(* CoDeSys 2.3 export: V4620699.EXP *)
(* Libraries: STANDARD.LIB 5.6.98 12:03:02, TcBase.lib 14.5.09 12:14:08, TcBaseMath.lib 27.7.04 12:07:56, TcCX1000System.lib 11.10.10 12:52:26, TcDrive.lib 25.1.17 09:42:28, TcEtherCAT.lib 30.11.16 19:52:18, TcIoFunctions.lib 27.1.17 17:22:22, TcMath.lib 23.9.04 15:15:30, TcMC.lib 27.7.15 08:51:38, TcNC.lib 10.10.08 17:55:34, TcNcDrive.lib 19.1.10 10:33:24, TcSystem.lib 7.6.16 11:01:22, TcTestAndSet.lib 23.2.09 12:50:08, TcUtilities.lib 3.2.16 16:08:58 *)

(* Task configuration *)
TASK Standard (PRIORITY := 0, INTERVAL := T#1ms);
PRG_STARTUP();
PRG_ERROR_WARNING_CTRLE();
PRG_VISU();
PRG_PROCESS();
PRG_STATION_WORK_ST1();
PRG_COLLISION_DETECTION();
PRG_VELOCITY_DETECTION();
PRG_HW_WORK_ST1();
PRG_HW_GENERAL();
END_TASK
TASK Ctrl_Panel (PRIORITY := 1, INTERVAL := T#100ms);
PRG_USB_IO_PANEL();
END_TASK

(* Global variable list: Constant_Variablen *)
VAR_GLOBAL CONSTANT
(*Constant variables Axis*)
	gciAxisZ_St1				:UINT:=1;
	gciAxisS_St1				:UINT:=2;
	gciAxisMax				:UINT:=2;

	gciStationSt1				:UINT:=1;

	(* developpement *)
	(*sRootPLC:STRING(255):='C:';*)
	(* machine *)
	cssRootPLC:STRING(255):='c:\';
	cssRootUSB:STRING(255):='d:\';
	(* HDD *)
	csiMaxFileLine:INT:=2230;
	csiMaxCharPerLine:INT:=135;
	(* Axis *)
	csiMaxAxisFileObj:INT:=50;
(* Visualisation number max page *)
	csiMaxPage:INT:=60;
	(* Profile *)
	csiMaxProfile:INT:=100;
	csiMaxProfileParameter:INT:=88;		(* BEF alt: 85 *) (* PUM alt: 78 *) (* PUM alt: 75 *) (* PUM alt: 61 *) (* PUM alt: 60 *) (* PUM alt: 53 *) (* IGS3 alt: 42 *)(* IGS2 alt: 38 *)(* IGS alt 36 *)
(* Page number definition *)
	gT_PageNumber:ST_VISUPAGENUMBER;
(* Anzahl maximal Wstk für Aufzeichnung *)
	ciMaxWP:INT:=100;
(* Max Anzahl Profilparameter *)
	ciMaxProfileParameter:INT:=1000;
(* Drehrichtung des Tellers *)
	gciModuloDirection:INT:=MC_Shortest_Way;

(* Skalierungswert für S Achse *)
	grScaleSAxis_Distance_SM:REAL:=966.0;
	grScaleSAxis_Speed_SM:REAL:=650;
	grMaxSAxis_Speed_SM:REAL:=8241.758;	(* Max Motor Drehzahl *)
	grScaleSAxis_Distance_L:REAL:=966.0;
	grScaleSAxis_Speed_L:REAL:=16;


	grMaxSAxis_Speed_L:REAL:=3000.0;		(* Max Motor Drehzahl *)	(* IGS angepasst *)
	grMaxSAxis_Speed_M:REAL:=6000.0;	(* Max Motor Drehzahl *)	(* IGS *)


(* ZUM LOESCHEN *)
	grScaleSAxis_Distance:REAL:=966.0;
	grScaleSAxis_Speed:REAL:=164;
	grMaxSAxis_Speed:REAL:=10000.0;			(* Max Motor Drehzahl *)
	grMaxSAxis_SpeedAllowed:REAL:=7000.0;	(* Max Motor Drehzal die für Maschine zugelassen ist *)
END_VAR

(* Global variable list: Globale_Variablen *)
VAR_GLOBAL
	QVisCtrl :ST_QVISCTRLE;(*~	(QVis) (InOut:2)	~*)
	T_ExchgParam :ST_QVIS_EXCHG_PARAM;(*~	(QVis) (InOut:2)	~*)
	T_VisuQVis:ST_QVIS;
	TProcess : ST_PROCESS;
	TStation_Work_St1 : ST_STATION;

(* Structure layer 2 *)
	T_CtrlePanel:ST_CTRLEPANEL;
	T_HDD:ST_HDD;
	T_NovRam : ST_NOVRAM;
(* StartUp *)
	T_StartUp:ST_STARTUP;
(* UPS *)
	T_CtrleUPS : ST_CTRLE_UPS;
	TStatusUPS:ST_UPSStatus;
(* Profile, 40 records ID for each Station *)
	T_Profile:ST_PROFILE;
(* TwinSAFE *)
	T_TwinSafeCtrleIN AT %I*:ST_TWINSAFE_CTRLE_IN;
	T_TwinSafeCtrleOUT AT %Q*:ST_TWINSAFE_CTRLE_OUT;
	T_TwinSafeIn AT %I*:ST_TWINSAFE_IN;
	T_TwinSafeOut AT %I*:ST_TWINSAFE_OUT;
	T_TwinSafeFBError AT %I*:ST_TWINSAFE_FB_ERROR;
	T_TwinSafe_Ctrle_Z_Axis_St1 AT %Q* : ST_TWINSAFE_DRIVE;
	T_TwinSafe_Status_Z_Axis_St1 AT %I* : ST_TWINSAFE_DRIVE;
	T_TwinSafe_Ctrle_S2_Axis_St1 AT %Q* : ST_TWINSAFE_DRIVE;		(* IGS *)
	T_TwinSafe_Status_S2_Axis_St1 AT %I* : ST_TWINSAFE_DRIVE;		(* IGS *)
	T_TwinSafe_Ctrle_S3_Axis_St1 AT %Q* : ST_TWINSAFE_DRIVE;		(* IGS *)
	T_TwinSafe_Status_S3_Axis_St1 AT %I* : ST_TWINSAFE_DRIVE;		(* IGS *)
	gT_SafetyStatus:ST_SAFETY_STATUS;

	T_Z_St1_Ctrle:ST_AXIS_CTRLE;
(* Static Error List *)
	T_ErrorList:ST_ERROR_LIST;	(* Static define Error List *)
(* Password *)
	T_Password:ST_PASSWORD;
(* Einrichtlampe *)
	TMachineLamp : ST_CYLINDER;
(* Control Button Start/Stop *)
	T_CtrleBtStartStop:ST_CTRLEBUTTON;
(* Kollisionsüberwachung *)
	TCollisionDetection:ST_COLLISION_DETECTION;
(* Status der Beckhoffklemmen und Kopplert *)
	T_TerminalState AT %I* :ST_TERMINAL_STATE;
(* Zähler für das Löschen der Vorwarnungen *)
	giDeleteMessageNumber: INT:=0;
	gcarAxisConfig		:ARRAY[1..gcIAxisMax] OF ST_EXCHG_PARAM_TEACHIN;
	gxHardwareOFF:BOOL;	(* Für Simulationszwecke ohne Hardware *)
	gxAxisOFF:BOOL;		(* Für Simulationszwecke wenn nur der Servocontroller der Z Achse fehlt und der Rest der Hardware vorhanden ist *)

(* Freigaben der Achsenbewegung mittels dem Joystick *)
	gxEnable_Joystick_Axis_Z:BOOL;
	gxReleaseEnableSwitch:BOOL;	(* Freigabe für Bewegung der Achsen mittels dem Zustimmschalter *)
	gxResetDataAnalysis_St1:BOOL;
	gxInitialStateActivated:BOOL;	(* Merker für Grundstellungsfahrt, ob dies ausgelöst wurde oder nicht *)
	gxAxisPositionSettled:BOOL;
	gxSetSpeedInMovement:BOOL;
	gxSetupFunctionActive:BOOL;
	gxAxisAbsolutMovementActive:BOOL;
	gxHandModeActive:BOOL;
	gxBlockSetQuality:BOOL;
	gxSpindelCalibrationONOFF_St1:BOOL;

	gT_PreWarning:ST_PREWARNING;

	gxAddInfeedZ:BOOL;
	gxSetPartQuality:BOOL;

	gxWP_Analyse_ActiveWork:BOOL;
	gxWP_Analyse_ActiveInfeed:BOOL;
	gxWP_Analyse_ActiveCentering:BOOL;
	gxWP_Analyse_ResetCentCountValue:BOOL;

	gdiSavePartQuality:DINT;

	gxMachineAutomodeActive_St1St2:BOOL;

(* Process Daten Aufzeichnung *)
	T_ProcessData_St1:ST_PROCESSDATA;

	gsDriveNameProcessData: STRING:='';

	gxBlockChangeMovementVisuActiveMessage:BOOL;

	gxSpindleOverloadError:BOOL;

	garRockerMeasureValue:ARRAY [1..200] OF REAL;
	grRockerMaxValue:REAL;
	grRockerMinValue:REAL;
	grRockerQuality:REAL;
	grRockerAmplitude:REAL;
	grRockerAmplitudeMin:REAL;
	grRockerAmplitudeMax:REAL;
	grRockerQualityMin:REAL;
	grRockerQualityMax:REAL;
	gdiRockerCountHC:DINT;
	gdiRockerCountHCTime:DINT;
	grRockerPosition:REAL;

	(* Globale Z Achsen Position *)
	grZ_LoadPos:REAL;
	grZ_WorkStartPos:REAL;
	grZ_WorkEndPos:REAL;

	gudiTorqueOverloadCounterValueSt1:UDINT;		(* IGS *)

	gxCentringActive:BOOL;						(* IGS3 *)
	gxOnlyCentringActive:BOOL;					(* IGS3 *)
	gxSuspensionONOFF:BOOL;					(* IGS3 *)

	garPositionEndProcCalc:ARRAY [1..1] OF REAL;
	garCentringEndProcCalc:ARRAY [1..1] OF REAL;
	gxZAxisVelocityCtrlActive:BOOL;
	gxZFollowDistanceError:BOOL;

	gxProcessCylindricalAreaActive:BOOL;
END_VAR

(* Global variable list: HW_IN_OUT *)
VAR_GLOBAL
(*++++++++++++++++++INPUT+++++++++++++++++++++++++++++*)
(*Local Inputs Schaltschrank*)
	IiAToolTorque_St1							AT%IB0		:INT;	(* Analoger Sensor für Drehmomentüberwachung für die Werkzeug Spindel *)
	IiASpeedServoDrive							AT%IB2		:INT;	(* Geschwindigkeitseinstellung der Achse Z1 *)
	IiAToolTorque2_St1							AT%IB4		:INT;	(* Analoger Sensor für Drehmomentüberwachung für die Werkzeug Spindel *)		(* IGS *)
	IiARes83										AT%IB6		:INT;	(* Reserve *)

	IxAirSupply									AT%IX8.0	:BOOL;	(* Ueberwacht den Mindestdruck des pneu.Netzes *)
	IxCabinDoorLocked							AT%IX8.1	:BOOL;	(* Kabinentüre (Sicherheitstüre) verriegelt *)
	IxStartButton									AT%IX8.2	:BOOL;	(* Externe Starttaste *)
	IxStopButton									AT%IX8.3	:BOOL;	(* Externe Stopptaste *)
	IxReleaseButton								AT%IX8.4	:BOOL;	(* Externe Freigabetaste für Energieversorgung *)
	IxRes105										AT%IX8.5	:BOOL;	(* Reserve *)
	IxJoystick_X_Plus								AT%IX8.6	:BOOL;	(* Joystick X Plus Jog Bewegung *)
	IxJoystick_X_Minus							AT%IX8.7	:BOOL;	(* Joystick X  negativ Ink Bewegung *)
	IxJoystick_Y_Plus								AT%IX9.0	:BOOL;	(* Joystick Z1 Achsenbewegung positiv *)
	IxJoystick_Y_Minus							AT%IX9.1	:BOOL;	(* Joystick Z1 Achsenbewegung negativ *)
	IxFuse24VDC_OK								AT%IX9.2	:BOOL;	(* Sicherungen 24VDC OK *)
	IxEnablingSwitchPlusButton						AT%IX9.3	:BOOL;	(* Zustimmschalter Plus Taste *)
	IxEnablingSwitchMinusButton					AT%IX9.4	:BOOL;	(* Zustimmschalter Minus Taste *)
	IxToolDeflection_St1							AT%IX9.5	:BOOL;	(* Überwachung der Werkzeug Auslenkung für die Werkzeug Spindel *)
	IxBrakeReleaseZ1Axis_St1						AT%IX9.6	:BOOL;	(* Sensor für Bremse gelöst bei der Z1 Achse (Hubachse) *)
	IxJoystick_WorkpieceClamp_ON_St1				AT%IX9.7	:BOOL;	(* Joystick für das einschalten der Werkstückfixierung *)
	IxJoystick_AirTable_ON						AT%IX10.0	:BOOL;	(* Joystick für das einschalten der Luft des Tisches	 *)
	IxJoystick_VaccumTable_ON					AT%IX10.1	:BOOL;	(* Joystick für das einschalten des Vakuums des Tisches *)
	IxUpperToolGuide_WorkpieceClamped_St1		AT%IX10.2	:BOOL;	(* Sensor für Überwachung der Werkstückfixierung *)
	IxToolSpindle_L_Connect_St1					AT%IX10.3	:BOOL;	(* Spindelkopf L angeschlossen-->Nur als Option vorgesehen: noch nichts unternehmen *)	(* INFO brauchts nicht, wird über Visu gemacht *)
	IxCylWPUnfixAtWorkPos_St1					AT%IX10.4	:BOOL;	(* Sensor für WstkEntspannen ist auf ArbeitsPosition *)							(* IGS3 *)
	IxToolDeflection2_St1							AT%IX10.5	:BOOL;	(* Überwachung der Werkzeug Auslenkung2 für die Werkzeug Spindel *)			(* IGS3 *)
	IxSuspenstionFilled							AT%IX10.6	:BOOL;	(* Sensor für Suspension ist gefüllt *)											(* IGS3 *)
	IxRes123										AT%IX10.7	:BOOL;	(* Reserve *)
	IxRes124										AT%IX11.0	:BOOL;	(* Reserve *)
	IxRes125										AT%IX11.1	:BOOL;	(* Reserve *)
	IxRes126										AT%IX11.2	:BOOL;	(* Reserve *)
	IxRes127										AT%IX11.3	:BOOL;	(* Reserve *)
	IxRes128										AT%IX11.4	:BOOL;	(* Reserve *)
	IxRes129										AT%IX11.5	:BOOL;	(* Reserve *)
	IxRes130										AT%IX11.6	:BOOL;	(* Reserve *)
	IxRes131										AT%IX11.7	:BOOL;	(* Reserve *)

	IxTorqueOverload_St1							AT%IX12.0	:BOOL;	(* Clock-->Signal induktiver Sensor für Drehmomentüberlast *)						(* IGS *)

(*++++++++++++++++++++++++++++
	Schnittstelle PLC to Safety Program:
++++++++++++++++++++++++++++*)
	IxTwinSafeQuickStopMaster1_1					AT%IX14.0	:BOOL;	(* QuickStop Achsen Mastermodul1_1 von TwinSAFE *)
	IxTwinSafeQuickStopMaster2_1					AT%IX14.1	:BOOL;	(* QuickStop Achsen Mastermodul2_1 von TwinSAFE *)							(* IGS *)
	IxTwinSafeQuickStopMaster2_2					AT%IX14.2	:BOOL;	(* QuickStop Achsen Mastermodul2_2 von TwinSAFE *)							(* IGS *)



(*++++++++++++++++++OUTPUT+++++++++++++++++++++++++++++*)
(*Local Outputs Schaltschrank*)
	QxCtrlLampStartButton							AT%QX0.0	:BOOL;	(* Kontroll LED externe Starttaste *)
	QxCtrlLampStopButton							AT%QX0.1	:BOOL;	(* Kontroll LED externe Stopptaste *)
	QxCtrlLampReleaseButton						AT%QX0.2	:BOOL;	(* Kotroll LED externe Freigabetaste für Energieversorgung *)
	QxCtrlLampAxesCurrentOff						AT%QX0.3	:BOOL;	(* Kontroll LED externe Ausschalttaste der Achsen Energieversorgung *)
	QxRes154									AT%QX0.4	:BOOL;	(* Reserve *)
	QxSignalLampGreen							AT%QX0.5	:BOOL;	(* Grüne Signallampe *)
	QxSignalLampRed							AT%QX0.6	:BOOL;	(* Rote Signallampe *)
	QxSignalLampYellow							AT%QX0.7	:BOOL;	(* Gelbe Signallampe *)
	QxCabinDoorLock								AT%QX1.0	:BOOL;	(* Verriegelungschalter der Kabinentüre, mit Magnetkraft *)
	QxSetupModeLamp							AT%QX1.1	:BOOL;	(* Gelbe Anzeige für den Einrichtbetrieb *)
	QxReadyToOperateMasterModul1				AT%QX1.2	:BOOL;	(* Betriebsbereitschaftsausgabe an Z1 *)
	QxEnablingSwitchVibration						AT%QX1.3	:BOOL;	(* Vibration des Zustimmschalter *)
	QxReadyToOperateMasterModul2				AT%QX1.4	:BOOL;	(* Betriebsbereitschaftsausgabe an S	ReadyToOperate to S *)					(* IGS *)
	QxMeasRangeTorqueSensor_St1				AT%QX1.5	:BOOL;	(* Drehmoment Sensor Bereichsumschaltung von 0-2Nm auf 0-0.5Nm Station 1 *)		(* IGS *)
	QxControlTorqueSensor_St1					AT%QX1.6	:BOOL;	(* Drehmoment Sensor Kontrollfunktion aktivieren Station 1 *)						(* IGS *)
	QxRes165									AT%QX1.7	:BOOL;	(* Reserve *)

	QxEnableQuickStopMasterModul1				AT%QX2.0	:BOOL;	(* Mastermodul für Z1 Achse aktivieren und einleiten des Schnellstop *)
	QxEnableQuickStopMasterModul2				AT%QX2.1	:BOOL;	(* Mastermodul für S Achse aktivieren und einleiten des Schnellstop *)				(* IGS *)
	QxCoolant_St1								AT%QX2.2	:BOOL;	(* Elektromagnetisches Ventil für Kühlmittel *)									(* IGS2 *)
	QxFastStrokeOn_St1							AT%QX2.3	:BOOL;	(* Schnellhub (Frequenzumformer) Ein *)										(* IGS2 *)
	QxRes214									AT%QX2.4	:BOOL;	(* Reserve *)
	QxRes215									AT%QX2.5	:BOOL;	(* Reserve *)
	QxRes216									AT%QX2.6	:BOOL;	(* Reserve *)
	QxRes217									AT%QX2.7	:BOOL;	(* Reserve *)
	QxRes218									AT%QX3.0	:BOOL;	(* Reserve *)
	QxRes219									AT%QX3.1	:BOOL;	(* Reserve *)
	QxRes220									AT%QX3.2	:BOOL;	(* Reserve *)
	QxRes221									AT%QX3.3	:BOOL;	(* Reserve *)
	QxRes222									AT%QX3.4	:BOOL;	(* Reserve *)
	QxRes223									AT%QX3.5	:BOOL;	(* Reserve *)
	QxRes224									AT%QX3.6	:BOOL;	(* Reserve *)
	QxRes225									AT%QX3.7	:BOOL;	(* Reserve *)

	QxMachineLamp								AT%QX4.0	:BOOL;	(* Maschinenleuchte *)
	QxRes201									AT%QX4.1	:BOOL;	(* Reserve *)
	QxRes202									AT%QX4.2	:BOOL;	(* Reserve *)
	QxRes203									AT%QX4.3	:BOOL;	(* Reserve *)

	QiAToolDeflection_SM_St1						AT%QB6	:INT;	(* Servoventil für Werkzeug Auslenkung der Werkzeug Spindel SM & M *)
	QiAToolTorqueHC_SM_St1						AT%QB8	:INT;	(* Servoventil für Drehmomentüberwachung HC des Spindelkopf SM *)		(* TODO löschen *)
	QiAToolTorqueOverload_SM_St1				AT%QB10	:INT;	(* Servoventil für Werkzeug Auslenkung der Werkzeug Spindel L *)		(* ALT: Servoventil für Drehmomentüberwachung Überlast des Spindelkopf SM *)
	QiAFastStroke								AT%QB12	:INT;	(* Analog Ausgang für FU (Schnellhub) *)										(* IGS2 *)
	QiARes254									AT%QB14	:INT;	(* Reserve *)
	QiARes255									AT%QB16	:INT;	(* Reserve *)
	QiARes256									AT%QB18	:INT;	(* Reserve *)
	QiARes257									AT%QB20	:INT;	(* Reserve *)

(* External Outputs at SMC Valve Block  *)
	Qby0ValveBlock								AT%QB30	:BYTE;	(* Byte 0 for Ethercat ValveBlock, Contains all following BOOL-Vars *)
	QxCylBrakeReleaseZAxis_Open_St1				AT%QX30.0	:BOOL;	(* Ventil für Bremszylinder der Z1 Achse für Bremse lösen *)
	QxCylBrakeReleaseZAxis_Close_St1			AT%QX30.1	:BOOL;	(* Ventil für Bremszylinder der Z1 Achse für Bremse aktivieren *)
	QxCylWorkpieceClamp_St1						AT%QX30.2	:BOOL;	(* Ventil für Werkstückfixierzylinder *)
	QxRes303									AT%QX30.3	:BOOL;	(* Reserve *)
	QxAirTable									AT%QX30.4	:BOOL;	(* Ventil für die Luft des Tisches *)
	QxRes305									AT%QX30.5	:BOOL;	(* Reserve *)
	QxVacuumTable								AT%QX30.6	:BOOL;	(* Ventil für das Vakuum des Tisches *)
	QxRes307									AT%QX30.7	:BOOL;	(* Reserve *)

	Qby1ValveBlock								AT%QB31	:BYTE;	(* Byte 1 for Ethercat ValveBlock, Contains all following BOOL-Vars *)
	QxCylWPUnfix_St1							AT%QX31.0	:BOOL;	(* Ventil für ZylWstkEntspannen *)											(* IGS3 *)
	QxRes309									AT%QX31.1	:BOOL;	(* Reserve *)
	QxCylStripperClose_St1						AT%QX31.2	:BOOL;	(* Ventil für ZylAbstreiferGeschlossen *)										(* IGS3 *)
	QxCylStripperOpen_St1						AT%QX31.3	:BOOL;	(* Ventil für ZylAbstreiferOffen *)												(* IGS3 *)
	QxRes312									AT%QX31.4	:BOOL;	(* Reserve *)
	QxRes313									AT%QX31.5	:BOOL;	(* Reserve *)
	QxRes314									AT%QX31.6	:BOOL;	(* Reserve *)
	QxRes315									AT%QX31.7	:BOOL;	(* Reserve *)

	Qby2ValveBlock								AT%QB32	:BYTE;	(* Byte 2 for Ethercat ValveBlock, Contains all following BOOL-Vars *)
	QxRes316									AT%QX32.0	:BOOL;	(* Reserve *)
	QxRes317									AT%QX32.1	:BOOL;	(* Reserve *)
	QxRes318									AT%QX32.2	:BOOL;	(* Reserve *)
	QxRes319									AT%QX32.3	:BOOL;	(* Reserve *)
	QxRes320									AT%QX32.4	:BOOL;	(* Reserve *)
	QxRes321									AT%QX32.5	:BOOL;	(* Reserve *)
	QxRes322									AT%QX32.6	:BOOL;	(* Reserve *)
	QxRes323									AT%QX32.7	:BOOL;	(* Reserve *)

(*++++++++++++++++++++++++++++
	Schnittstelle PLC to Safety Program:
++++++++++++++++++++++++++++*)
	QxTwinSafeReleaseButton						AT%QX35.0	:BOOL;	(* Output to safety prog *)
	QxTwinSafeServoDrivesRdy					AT%QX35.1	:BOOL;	(* Output to safety prog,ALL Servo-Controler: No Error *)

END_VAR

(* Global variable list: TwinCAT_Configuration *)
(* Generated automatically by TwinCAT - (read only) *)
VAR_CONFIG
	PRG_HW_WORK_ST1.IuiActualTorqueAxisZ_St1 AT %IB1656 : UINT;
	PRG_HW_WORK_ST1.IwInputState_Z_Axis_St1 AT %IB1658 : WORD;	(*  ~ {LinkedWith:TIID^Gerät 4 (EtherCAT)^Achse Z St1 (AX5106-0000-0210)^AT^Digital inputs, state} *)
	PRG_HW_WORK_ST1.IuiActualTorqueAxisS_St1 AT %IB1660 : UINT;
	PRG_HW_WORK_ST1.IwInputState_S1_Axis_St1 AT %IB1662 : WORD;
	PRG_HW_WORK_ST1.IwInputState_S2_Axis_St1 AT %IB1012 : WORD;	(*  ~ {LinkedWith:TIID^Gerät 4 (EtherCAT)^Antrieb S2 S3 St1 (AX5206-0000-0203)^AT 1^Digital inputs, state} *)
	PRG_HW_WORK_ST1.IwInputState_S3_Axis_St1 AT %IB1014 : WORD;	(*  ~ {LinkedWith:TIID^Gerät 4 (EtherCAT)^Antrieb S2 S3 St1 (AX5206-0000-0203)^AT 2^Digital inputs, state} *)
	PRG_HW_WORK_ST1.stZRefIn_St1 AT %IB1016 : NCTOPLC_AXLESTRUCT;	(*  ~ {LinkedWith:TINC^NC-Task 1 SAF^Achsen^Achse Z^Ausgänge^Achse Z_ToPlc} *)
	PRG_HW_WORK_ST1.stZRefOut_St1 AT %QB10012 : PLCTONC_AXLESTRUCT;	(*  ~ {LinkedWith:TINC^NC-Task 1 SAF^Achsen^Achse Z^Eingänge^Achse Z_FromPlc} *)
	PRG_HW_WORK_ST1.stZDriveState_St1 AT %IB1144 : ST_AXIS_DRIVESTATE;
	PRG_HW_WORK_ST1.stSRefIn_St1 AT %IB1148 : NCTOPLC_AXLESTRUCT;	(*  ~ {LinkedWith:TINC^NC-Task 1 SAF^Achsen^Achse S1^Ausgänge^Achse S1_ToPlc} *)
	PRG_HW_WORK_ST1.stSRefOut_St1 AT %QB10140 : PLCTONC_AXLESTRUCT;	(*  ~ {LinkedWith:TINC^NC-Task 1 SAF^Achsen^Achse S1^Eingänge^Achse S1_FromPlc} *)
	PRG_HW_WORK_ST1.stS2RefIn_St1 AT %IB1276 : NCTOPLC_AXLESTRUCT;	(*  ~ {LinkedWith:TINC^NC-Task 1 SAF^Achsen^Achse S2^Ausgänge^Achse 2_ToPlc} *)
	PRG_HW_WORK_ST1.stS2RefOut_St1 AT %QB10268 : PLCTONC_AXLESTRUCT;	(*  ~ {LinkedWith:TINC^NC-Task 1 SAF^Achsen^Achse S2^Eingänge^Achse 2_FromPlc} *)
	PRG_HW_WORK_ST1.stS3RefIn_St1 AT %IB1404 : NCTOPLC_AXLESTRUCT;	(*  ~ {LinkedWith:TINC^NC-Task 1 SAF^Achsen^Achse S3^Ausgänge^Achse 3_ToPlc} *)
	PRG_HW_WORK_ST1.stS3RefOut_St1 AT %QB10396 : PLCTONC_AXLESTRUCT;	(*  ~ {LinkedWith:TINC^NC-Task 1 SAF^Achsen^Achse S3^Eingänge^Achse 3_FromPlc} *)
	PRG_HW_WORK_ST1.stBubblerDataINSt1 AT %IB1648 : ST_COMM_IN_DCAXIS;
	PRG_HW_WORK_ST1.stBubblerDataOUTSt1 AT %QB10587 : ST_COMM_OUT_DCAXIS;
	PRG_HW_WORK_ST1.stFeedpumpINDataSt1 AT %IB1651 : ST_COMM_IN_DCAXIS;
	PRG_HW_WORK_ST1.stFeedpumpOUTDataSt1 AT %QB10590 : ST_COMM_OUT_DCAXIS;
	PRG_HW_WORK_ST1.IudiTorqueOverloadCounterValue_St1 AT %IB1532 : UDINT;	(*  ~ {LinkedWith:TIID^Gerät 1 (EtherCAT)^E-CAT Netzteil  (EK1200)^Zaehlerklemme 15 (EL1502)^CNT Inputs^Counter value} *)
	PRG_USB_IO_PANEL.IarxCtrlePanelButton AT %IB1536 : ARRAY [1..10] OF BOOL;
	PRG_USB_IO_PANEL.QarxCtrlePanelLed AT %QB10524 : ARRAY [1..10] OF BOOL;
	.T_TwinSafeCtrleIN AT %IB1546 : ST_TWINSAFE_CTRLE_IN;
	.T_TwinSafeCtrleOUT AT %QB10534 : ST_TWINSAFE_CTRLE_OUT;
	.T_TwinSafeIn AT %IB1549 : ST_TWINSAFE_IN;
	.T_TwinSafeOut AT %IB1569 : ST_TWINSAFE_OUT;
	.T_TwinSafeFBError AT %IB1577 : ST_TWINSAFE_FB_ERROR;
	.T_TwinSafe_Ctrle_Z_Axis_St1 AT %QB10536 : ST_TWINSAFE_DRIVE;
	.T_TwinSafe_Status_Z_Axis_St1 AT %IB1585 : ST_TWINSAFE_DRIVE;
	.T_TwinSafe_Ctrle_S2_Axis_St1 AT %QB10553 : ST_TWINSAFE_DRIVE;
	.T_TwinSafe_Status_S2_Axis_St1 AT %IB1602 : ST_TWINSAFE_DRIVE;
	.T_TwinSafe_Ctrle_S3_Axis_St1 AT %QB10570 : ST_TWINSAFE_DRIVE;
	.T_TwinSafe_Status_S3_Axis_St1 AT %IB1619 : ST_TWINSAFE_DRIVE;
	.T_TerminalState AT %IB1636 : ST_TERMINAL_STATE;
END_VAR

(* Data type in Axis/Axis_DC_KL2552 *)
TYPE ST_AXIS_FILE_OBJ_DCAXIS :
STRUCT
	sData: ARRAY[1..csiMaxAxisFileObj] OF STRING(80);
END_STRUCT
END_TYPE

(* Data type in Axis/Axis_DC_KL2552 *)
TYPE ST_COMM_IN_DCAXIS :
STRUCT
	usiStatusWord :USINT;
	iDataIn :INT;
END_STRUCT
END_TYPE

(* Data type in Axis/Axis_DC_KL2552 *)
TYPE ST_COMM_OUT_DCAXIS :
STRUCT
	usiControlWord :USINT;
	iDataOut :INT;
END_STRUCT
END_TYPE

(* Data type in Axis/Axis_DC_KL2552 *)
TYPE ST_CONFIG_GENERAL_DCAXIS :
STRUCT
	sDeviceName:STRING(32);
	sDeviceFileName:STRING(32);
	sServoNetId:STRING(23);		(* Beckhoff *)
	udiNodeId:UDINT;				(* Maxon *)
	iTyp:INT;
	lrScaleFactor:LREAL:=0.0;
	lrInitFactor:LREAL:=0.0;
END_STRUCT
END_TYPE

(* Data type in Axis/Axis_DC_KL2552 *)
TYPE ST_CONFIG_OBJECT_DCAXIS :
STRUCT
	diMaxMotorCurrent:DINT:=0;
	diNominalMotorCurrent:DINT:=0;
	diMotorResistor:DINT:=0;
	diKpSpeedControl:DINT:=0;
	diTnCurrentControl:DINT:=0;
	diMaxTorqueMotor:DINT:=0;
	xSpeedControlAcitv:BOOL:=FALSE;
	xCurrentControlAcitv:BOOL:=FALSE;
	xWinCurrentControlActiv:BOOL:=FALSE;
	xTorqueControlAcitv:BOOL:=FALSE;
	xOverVoltageActiv:BOOL:=FALSE;
END_STRUCT
END_TYPE

(* Data type in Axis/Axis_DC_KL2552 *)
TYPE ST_CTRLE_DCAXIS :
STRUCT
(* Input *)
	xExecute:BOOL:=FALSE;
	iFunction:INT:=0;
	xReset:BOOL:=FALSE;
	lrVelocity:LREAL:=0;
	tAcceleration:TIME:=T#0s;
	tDecceleration:TIME:=T#0s;
	iRegisterNr:INT:=0;
	iValueRegister:INT:=0;

(* Output *)
	xDone:BOOL:=FALSE;
	xErr:BOOL:=FALSE;
	udiErrorID:UDINT:=0;
	xPower:BOOL:=FALSE;
	xReady:BOOL:=FALSE;
	xNotMoving:BOOL:=FALSE;
END_STRUCT
END_TYPE

(* Data type in Axis/Axis_DC_KL2552 *)
TYPE ST_DC_AXIS :
STRUCT
	T_CtrleDCAxis : ST_CTRLE_DCAXIS;
	T_ParamFileObj:ARRAY[1..20] OF ST_PARAM_FILE_OBJ_DCAXIS;
	T_Config_Gen:ST_CONFIG_GENERAL_DCAXIS;
	T_Config_ObjFileValue:ST_CONFIG_OBJECT_DCAXIS;
	T_FileObj:ST_AXIS_FILE_OBJ_DCAXIS;
END_STRUCT
END_TYPE

(* Data type in Axis/Axis_DC_KL2552 *)
TYPE ST_PARAM_FILE_OBJ_DCAXIS :
STRUCT
	iRegisterNr:INT:=0;
	iBitValue:INT:=0;
	lrReal:LREAL:=0;
	sName:STRING(20);
END_STRUCT
END_TYPE

(* Data type in Axis *)
TYPE ST_AXIS :
STRUCT
	T_CtrleSingle:ST_CTRLESINGLE;
	T_CtrleMulti:ST_CTRLEMULTI;
	T_ParamFileObj:ARRAY[1..40] OF ST_PARAM_FILE_OBJ;
	T_Config_Gen:ST_CONFIG_GENERAL;
	T_Config_ObjFileValue:ST_CONFIG_OBJECT;
	T_Config_Setting:ST_CONFIG_SETTING;
	T_LiveValue:ST_LIVEVALUE;
	T_Oscillation:ST_OSCILLATION;
	T_FileObj:ST_AXIS_FILE_OBJ;
	T_DriveState:ST_AXIS_DRIVESTATE;
END_STRUCT
END_TYPE

(* Data type in Axis *)
TYPE ST_AXIS_CTRLE :
STRUCT
	diVelocityCommandValue AT %QD1000	:DINT;	(* Verknüpfung mit E/A Ebene des Servos der Z Achse *)
	nOutData2 AT %ID1003 :ARRAY [0..1] OF UINT;	(* Verknüpfung mit NC Ebene des Servos der Z Achse *)
END_STRUCT
END_TYPE

(* Data type in Axis *)
TYPE ST_AXIS_DRIVESTATE :
STRUCT
	usiDriveState0:USINT;
	usiDriveState1:USINT;
	usiDriveState2:USINT;
	usiDriveState3:USINT;
END_STRUCT
END_TYPE

(* Data type in Axis *)
TYPE ST_AXIS_FILE_OBJ :
STRUCT
	sData: ARRAY[1..csiMaxAxisFileObj] OF STRING(80);
END_STRUCT
END_TYPE

(* Data type in Axis *)
TYPE ST_AXIS_LIVESTATE : (*Axis State struct  for HMI-Interface*)
STRUCT
	rActPos				:REAL;	(*PLC To HMI:actual position*)
	rActSpeed			:REAL;	(*PLC To HMI:actual speed*)
	bActState			:BYTE;	(*PLC To HMI:actual state*)
	rTeachPosStored		:REAL;	(*PLC To HMI:stored position according 'iTeachSelPos' *)
	rSWLimPos			:REAL;	(*SW-Limit positive value, Grenzwerte für HMI-Eingabe *)
	rSWLimNeg			:REAL;	(*SW-Limit negative value,Grenzwerte für HMI-Eingabe*)

	rSetSpeed			:REAL;	(*HMI To PLC:new speed setpoint*)
	rSetPos				:REAL;	(*HMI To PLC:new position setpoint*)
	iTeachSelPos		:INT;	(*HMI To PLC:actual  selection 'teach-list' *)

	xAxisSelect			:BOOL;	(* Anzeigen welche Achse ausgewählt ist *)
END_STRUCT
END_TYPE

(* Data type in Axis *)
TYPE ST_CONFIG_GENERAL :
STRUCT
	sDeviceName:STRING(32);
	sDeviceFileName:STRING(32);
	sServoNetId:STRING(23);		(* Beckhoff *)
	sAmsNetId:T_AmsNetId;		(* Maxon *)
	udiNC_TaskIdxGrp:UDINT;		(* Beckhoff *)
	udiNodeId:UDINT;				(* Maxon *)
	iTyp:INT;
	wPosLimitSwitchBit:WORD;		(* Gilt nur für AX5xxx Antriebe und nur falls Endschalter belegt ist
								    Bei Single oder Dualservoantrieb gilt für Achse 1
									PosLimitSwitch:8
								    Bei Dualservoantrieb gilt für Achse 2
									PosLimitSwitch:32
								*)
	wNegLimitSwitchBit:WORD;		(* Gilt nur für AX5xxx Antriebe und nur falls Endschalter belegt ist
								    Bei Single oder Dualservoantrieb gilt für Achse 1
									NegLimitSwitch:16
								    Bei Dualservoantrieb gilt für Achse 2
									NegLimitSwitch:64
								*)
END_STRUCT
END_TYPE

(* Data type in Axis *)
TYPE ST_CONFIG_OBJECT :
STRUCT
(* Object value *)
	lrMaxVelocity:LREAL;
	lrCalVelocityForward:LREAL;
	lrCalVelocityBackward:LREAL;
	lrAcceleration:LREAL;
	lrDecceleration:LREAL;
	lrJerk:LREAL;
	xSWLimitPos:BOOL;
	lrSWLimitPos:LREAL;
	xSWLimitNeg:BOOL;
	lrSWLimitNeg:LREAL;
	lrScaleFactor:LREAL;
END_STRUCT
END_TYPE

(* Data type in Axis *)
TYPE ST_CONFIG_SETTING :
STRUCT
	lrJogFast:LREAL;
	lrJogSlow:LREAL;
	lrJogStepFast:LREAL;
	lrJogStepSlow:LREAL;
	lrVelocityAbs:LREAL;
	lrVelocityRel:LREAL;
	lrVelocityProcess:LREAL;
	lrSpindleCurrentLimit:LREAL;
	xHardwareLimitPos:BOOL;
	xHardwareLimitNeg:BOOL;
	xSoftwareLimitPos:BOOL;
	xSoftwareLimitNeg:BOOL;
	lrHWLimitDecceleration:LREAL;
	rHCRampDeceleration:REAL;
	rHCRampJerk:REAL;
	xAbsoluteEncoder:BOOL;
END_STRUCT
END_TYPE

(* Data type in Axis *)
TYPE ST_CTRLEMULTI :
STRUCT
(* Input *)
	xExecute:BOOL:=FALSE;
	xReset:BOOL:=FALSE;
	iNumerator:INT:=1;
	uiDenominator:UINT:=1;
	iFunction:INT:=0;

(* Ouput *)
	xDone:BOOL:=FALSE;
	xErr:BOOL:=FALSE;
	udiErrorID:UDINT:=0;
END_STRUCT
END_TYPE

(* Data type in Axis *)
TYPE ST_CTRLESINGLE :
STRUCT
(* Input *)
	xExecute:BOOL:=FALSE;		(* Ausführen einer Achsen Funktion *)
	iFunction:INT:=0;				(*
								1=Achse Resetten
								2=Achsen Datei lesen
								3=Achsenstrom Einschalten-->Drehmoment ON
								4=Achsenstrom Ausschalten-->Drehmoment OFF
								5=Achsenbewegung stoppen
									-->lrDecceleration und lrJerk übergeben
								6=Geschwindigkeitsbewegung-->Sobald Drehzahl erreicht wird, dann wird das Endflag xDone gesetzt
									-->lrVelocity, lrAcceleration, lrDecceleration und lrJerk übergeben
								7=Absolute Bewegung-->Erst wenn Position erreicht wird, dann wird das Endflag xDone gesetzt
									-->lrPosition, lrVelocity, lrAcceleration, lrDecceleration und lrJerk übergeben
								8=Relative Bewegung-->Erst wenn der Weg abgefahren ist, dann wird das Endflag xDone gesetzt
									-->lrDistance, lrVelocity, lrAcceleration, lrDecceleration und lrJerk übergeben
								9=Achse Referenzieren-->Erst wenn Achse Referenziert ist, dann wird das Endflag xDone gesetzt
									-->rSetPosition für den Referenzoffset übergeben (restliche Parameter erfolgt über NC Parameter)
								10=Overrider der Geschwindigkeit in %
									-->dwOverride übergeben (...0.9=90%, 1.0=100%, 1.1=110%...)
								11=Überschreiben der Aktuellen Position
									-->rSetPosition übergeben
								12=Während Achse in Bewegung ist (Geschwindigkeit, Absolut, Relativ oder Modulo) kann eine neue Geschwindigkeit vorgegeben werden
									-->lrVelocity übergeben
								13=Referenzflag Manuell setzten
								14=Referenzflag Manuell zurück setzen
								15=Einschalten des Externen Sollwertgenerator. Die Achse übernimmt anschliessend die Sollwertvorgaben aus ihrem zyklischen Achsinterface
								       (fExtSetPos, fExtSetVelo, fExtSetAcc, nExtSetDirection)
								16=Ausschalten des Externen Sollwertgenerator
								17=Einschalten einer Oszillationsbewegung
									folgende Parameter müssen übergeben werden:
									-->T_Oscillation.rFrequence: Oszillationsfrequenz
									-->T_Oscillation.rOffset: Oszillationshub (positiver Wert: erste Bewegung in positiver Richtung! negativer Wert: erste Bewegung in negativer Richtung 
									-->T_Oscillation.iCycle: Anzahl Oszillationsperioden
								18=Während einer Absoluten Positionierung kann eine neue Position vorgegeben werden
									-->lrPosition muss übergeben werden
								19=Berechnung, mittels Achsbewegung, des Winkels zwischen Ref.Sensor und EncoderIndex
								20=Setzen der Default Achsen Parameter an der Achsenstruktur
								21=Senden der Achsenparameter (eingelsen über die Datei oder Default Achsen Parameter) an die NC Parameter
								22=Senden eines String über den ADS um Zugriff direkt auf die Servo Parameter
									-->sSend übergeben
								23=Achsdatei erstellen mit den Achse Parameter (ist nicht implementiert)
								24=Modulo Bewegung für z.B. Tellerpositionen anzufahren
									-->lrPosition, lrVelocity, lrAcceleration, lrDecceleration und lrJerk übergeben
								25=Einschalten des Positiven Software Endschalter (Position muss im System Manager manuell eingetragen werden)
								26=Ausschalten des Positiven Software Endschalter
								*)
	xReset:BOOL:=FALSE;			(* Zurücksetzen des Achsen Treiberbausteins *)
	lrPosition:LREAL:=0;			(* Positionsübergabe für Absolut oder Modulo Bewegung *)
	lrDistance:LREAL:=0;			(* Streckenübergabe für Relative Bewegung *)
	lrVelocity:LREAL:=0;			(* Geschwindigkeit in Technische Einheit für jegliche Bewegungen *)
	lrAcceleration:LREAL:=0;		(* Positive Beschleunigung für jegliche Bewegungen *)
	lrDecceleration:LREAL:=0;		(* Negative Beschleunigung für jegliche Bewegungen und Stopp Rampe *)
	lrJerk:REAL:=0;				(* Ruck für jegliche Bewegungen und Stopp Rampe *)
	dwOverride:DWORD:=100;		(* Overrider der Geschwindigkeit in % --> ...0.9=90%, 1.0=100%, 1.1=110%... *)
	rSetPosition:REAL:=0;			(* Setzen der Position für Referenzoffset oder überschreiben der Aktuellen Position *)
	rSetTorque:REAL:=0;			(* Festlegen des Drehmomentes für Maxon Motoren *)
	sSend:STRING(20):='';			(* Senden eines String über das ADS für Servoparameter *)
	lrScaleFactor:LREAL:=0;		(* Skalierungsfaktor für Technische Einheit *)
	rNominalSpeed:REAL:=0;		(* Nenndrehzahl für Maxon Motoren *)
	iModuloDirection:INT;			(*	Enum Werte:
									MC_Positive_Direction := 1,
    									MC_Shortest_Way :=2,
    									MC_Negative_Direction :=3,
    									MC_Current_Direction :=4
								*)
	lrHardwarePosition:LREAL;		(* Gilt für Absolut Encoder *)
	xMoveAwayFromHWLimitSwitchActive:BOOL;	(* Gilt für AX5000 Servo: Mittels diesem Signal = TRUE--> ermöglicht es die Achse auf den Endschalter zu fahren und dass man es über die Steuerung
												wieder vom Endschalter wegfahren kann. Ist es FALSE, dann muss die Achse von Hand vom Endschalter weggezogen werden *)
	xAX5000Active:BOOL;			(* FALSE = AX25xx, TRUE = AX5xxx *)
	xKL2541Active:BOOL;			(* TRUE = Schrittmotor KL2541 *)
(* Output *)
	xDone:BOOL:=FALSE;			(* Nach dem starten der Funktion wird es zu FALSE und sobald die Funktion beendet wird dann wird es auf TRUE gesetzt!
					    	    		    sollte ein Fehler entstehen, dann bleibt es auf FALSE bis der Baustein zurückgesetzt wird *)
	xErr:BOOL:=FALSE;			(* Sollte bei einer Funktion ein Fehler entstehen, dann wird dieser Flag gesetzt-->In diesem Fall wird das xDone Flag nicht gesetzt *)
	udiErrorID:UDINT:=0;			(* Fehlernummer, falls des xErr Flag gesetzt wird
									Fehler aus der NC Ebene:
									0x40nn=Allgemeine NC-Fehler
									0x41nn=Kanalfehler
									0x42nn=Gruppenfehler
									0x43nn=Achsfehler
									0x44nn=Geberfehler
									0x45nn=Reglerfehler
									0x46nn=Antriebfehler
									0x4Ann=Tabellenfehler	
									0x4Bnn=NC-SPS-Fehler
									-->Genaueres entnehme man aus den TwinCAT NC Fehlercodes!
									Fehlernummer des Treibers:
									16#F000=Aufgerufene Funktionsnummer gibt es nicht
									16#F100=Während der Aktiven StoppFunktion wurde eine andere (Ausnahme Reset) Funktion aufgerufen
									16#F101=Beim senden der Achsenparameter Funktion ist ein Timeout entstanden beim ein- oder ausschalten des Achsenstromes
									16#F102=Beim einschalten des Positiven Software Endschalter darf die Achse sich nicht bewegen
									16#F103=Beim einschalten des Positiven Software Endschalter darf die Achse nicht im Slave Mode betrieben sein
									16#F104=Timeout für das lesen der Achsen Parameter Datei->T_HDD ist gesperrt
									16#F105=Timeout für das schreiben der Achsen Parameter Datei->T_HDD ist gesperrt
									16#F106=Beim senden eines Achsenstring Funktion ist der empfangene String nicht gleichwertig wie der gesendete String-->Bestätigung des Servos Misslungen
									16#F201=Achsen Parameter Datei nicht gefunden
									16#F202=Falscher Syntax für eingelesener Achsen Parameter Datei
								*)
	xPower:BOOL:=FALSE;			(* Zeigt den Status des Motorstromes an-->TRUE=Strom ON, FALSE=Strom OFF *)
	xReady:BOOL:=FALSE;		(* Zeigt den Status ob der Servo bereit steht oder nicht-->TRUE=Servo Bereit, FALSE=Servo nicht Bereit *)
	xNotMoving:BOOL:=FALSE;		(* Zeigt den Status ob die Achse sich bewegt-->TRUE=Achse steht still, FALSE=Achse bewegt sich *)
	xMovingForward:BOOL:=FALSE;		(* Zeigt den Status ob die Achse sich in Positiver Richtung bewegt-->TRUE=Achse bewegt sich in Positiver Richtung *)
	xMovingBackwards:BOOL:=FALSE;	(* Zeigt den Status ob die Achse sich in Negativer Richtung bewegt-->TRUE=Achse bewegt sich in Negativer Richtung *)
	xRef:BOOL:=FALSE;			(* Zeigt den Status ob die Achse referenziert ist oder nicht-->TRUE=Achse Referenziert, FALSE=Achse nicht Referenziert *)
	xSlave:BOOL:=FALSE;			(* Zeigt den Status ob die Achse als Slave bei Master/Slave Verbindung aktiv ist-->TRUE=mit einer anderen Achse gekoppelt als Slave, FALSE=Standalone Betrieb oder Master *)
	xConstantVel:BOOL:=FALSE;	(* Zeigt den Status ob bei Achsbewegung die vorgegebene Drehzahl erreicht wurde-->TRUE=Drehzahl erreicht, FALSE=Drehzahl nicht erreicht *)
	xBusyNewPosAndVel:BOOL:=FALSE;	(* Zeigt den Status ob neue Geschwindigkeit oder Position Aktiv ist-->TRUE=Neue Geschw./Pos ist in Bearbeitung, FALSE=Keine neue Geschw./Pos in Bearbeitung *)
	xDriveTorque:BOOL:=FALSE;	(* Zeigt ob die Achse in Drehmomentbetrieb ist-->gilt für Maxon Motoren *)
	xSWLimitPos:BOOL:=FALSE;	(* Definiert ob die Achse einen Positiven Software Endschalter hat *)
	xSWLimitNeg:BOOL:=FALSE;	(* Definiert ob die Achse einen Negativen Software Endschalter hat *)
	xHWLimitPos:BOOL:=FALSE;	(* Definiert ob die Achse einen Positiven Hardware Endschalter hat *)
	xHWLimitNeg:BOOL:=FALSE;	(* Definiert ob die Achse einen Negativen Hardware Endschalter hat *)
	xStateHWLimitPos:BOOL:=FALSE;	(* Zeigt den Status des Positiven Software Endschalter-->TRUE=SW_PLS ON, FALSE=SW_PLS OFF *)
	xStateHWLimitNeg:BOOL:=FALSE;	(* Zeigt den Status des Negativen Software Endschalter-->TRUE=SW_NLS ON, FALSE=SW_NLS OFF *)
	xStateSWLimitPos:BOOL:=FALSE;	(* Zeigt den Status des Positiven Hardware Endschalter-->TRUE=HW_PLS ON, FALSE=HW_PLS OFF *)
	xStateSWLimitNeg:BOOL:=FALSE;	(* Zeigt den Status des Negativen Hardware Endschalter-->TRUE=HW_NLS ON, FALSE=HW_NLS OFF *)
	xSpindleBlocked:BOOL:=FALSE;	(* Zeigt an ob die Spindel blockiert ist-->gilt für Maxon Motoren *)
	iZAngleRefIndex:INT;		(* Gilt für die Prozedur für das einstellen des Referenzindex der Achse-->Für die Visu damit der Winkel angezeigt werden kann zwischen RefSensor und EncoderIndex *)
	xSWLimitSwitchPosActivated:BOOL:=FALSE;	(* Zeigt den Status ob der Positive Software Endschalter gesetzt wurde oder nicht *)
	xSlowFast:BOOL:=TRUE;		(* Zeigt an ob die langsame/schnelle geschwindigkeit oder kurzes/langes Inkrement für INK/JOG Bewegung ausgewählt ist-->gilt nur für ausserhalb des Treiberbausteins
									FALSE=langsame Geschwindigkeit(JOG) oder kurzes Inkrement(INK) 
									TRUE=schnelle Geschwindigkeit(JOG) oder langes Inkrement(INK)
								*)
	xJogInc:BOOL;	(* Umschaltung zwischen Jog und Ink *)
	sDeviceName:STRING(255);	(* Beckhoff oder Maxon für das konvertieren der eingelesenen Achsendatei *)
	xAxisCollisionError:BOOL;
	xHomingSensor:BOOL;			(* TRUE= Referenzsensor ON *)

(* Für Maxon ESCON Servocontroller *)
	iMaxVelocty	:UINT;(*Maximum rpm*)
	xAmplReady		:BOOL;
	xAmplPower		:BOOL;
	xStandstill		:BOOL;
	xSpindleOverloadError:BOOL;
END_STRUCT
END_TYPE

(* Data type in Axis *)
TYPE ST_LIVEVALUE :
STRUCT
	dwState:DWORD;
	uiActualTorque:UINT;
	diActualTorqueCalc:DINT;	(* entsricht dem uiActualTorque, nur dass positiver und negativer Torque berücksichtigt wird *)
	lrActualVelocity:LREAL;
	lrActualPosition:LREAL;
	bDigitalInput:BYTE;
	lrSollPosition:LREAL;
	lrActualPositionNotModulo:LREAL;
	uiDigitalInput:UINT;
END_STRUCT
END_TYPE

(* Data type in Axis *)
TYPE ST_OSCILLATION :
STRUCT
	rFrequence:REAL;
	rOffset:REAL;
	rPosTorqueLimitOffset:REAL;
	iCycle:INT;
END_STRUCT
END_TYPE

(* Data type in Axis *)
TYPE ST_PARAM_FILE_OBJ :
STRUCT
	udiIdxGroup:UDINT:=0;
	udiIndexOffset:UDINT:=0;
	udiLength:UDINT:=0;
	lrReal:LREAL:=0;
	sName:STRING(20);
END_STRUCT
END_TYPE

(* Data type in CollisionDetection *)
TYPE ST_COLLISION_DETECTION :
STRUCT
(* Bearbeitungsstation *)
	xZAxisBrakeReleased:BOOL;
END_STRUCT
END_TYPE

(* Data type in Controller *)
TYPE ST_CTRL_PID_PARAM :
STRUCT
 	rCtrlCycleTime         : REAL;		(* Zykluszeit, mit der der Regelkreis bearbeitet wird. Der Funktionsbaustein berechnet mit dieser Eingangsgröße intern,
																	ob die Zustands- und Ausgangsgrößen im aktuellen Zyklus aktualisiert werden müssen. *)
 	rKp                    : REAL;					(* Reglerverstärkung / Reglerbeiwert *)
 	rKi                    : REAL; 			(* Nachstellzeit, wenn diese zu T#0s parametriert ist, wird der I-Anteil deaktiviert.*)
	rKd                    : REAL; 			(* Vorhaltzeit, wenn diese zu T#0s parametriert ist, wird der D-Anteil deaktiviert. *)
	rOutMaxLimit       : REAL;
 	rOutMinLimit         : REAL;
	xReset_I_Anteil:BOOL;
END_STRUCT
END_TYPE

(* Data type in Cylinder *)
TYPE ST_ANALOG :
STRUCT
(* input *)
	tDelayActiv:TIME;			(* Für die FunktionNr 2 lässt sich mittels dieser Zeit(falls <> 0s) die Impulsdauer festlegen, d.h. der Ausgang bleibt für diese Zeit gesetzt *)
	tDelayAfterSensor:TIME;	(* Für die FunktionNr 1 und 2 lässt sich mit Sensorüberwachung eine Zeit definieren welches nachdem der Sensor eintrifft bis das Flag xDone gesetzt wird *)
	iAnalogIN:INT;			(* Analog Wert 0 - 32767 (0 - 10V) welcher für den Ausgang übergeben wird *)
	rForceIn:REAL;			(* Technische Einheit-->wird intern im Zylinder Treiber nicht verwendet-->Ausserhalb muss die Umrechnung für den iAnalogIN erfolgen *)
	lrVoltageIN:LREAL;		(* Spannungswert in Volt (V) *)
	iRampFctOn:INT;			(* Rampe für FunktionNr 2 für das setzen des Analogen Ausganges
								1=Parabelfunktion
								2=e-Funktion
								3=Linearfunktion
							*)
	iRampFctOff:INT;			(* Rampe für FunktionNr 1 für das setzen des Analogen Ausganges
								1=Parabelfunktion
								2=e-Funktion
								3=Linearfunktion
							*)
	rStepValue:REAL;			(* Schrittgrösse für Rampe FunktionNr 1 und 2
							    	Wert 0 = Rampenfunktion ausgeschaltet
							*)
(* Output *)
	xActiv:BOOL;				(* Analogausgang = 0 --> FALSE
							    Analogausgang > 0 --> TRUE
							*)
	iAnalogOut:INT;			(* Analog Wert 0 - 32767 (0 - 10V) für Effektiven Wert welcher am Ausgang steht-->muss ausserhalb des Zylinder Treiber zugewiesen werden *)
	rForceOut:REAL;			(* Technische Einheit für Effektiven Wert welcher am Ausgang steht-->muss ausserhalb des Zylinder Treiber berechnet und zugewiesen werden *)
	rTorqueOut:REAL;			(* Technische Einheit für Effektiven Wert welcher am Ausgang steht-->muss ausserhalb des Zylinder Treiber berechnet und zugewiesen werden *)
	rPosOut:REAL;
	lrTorqueOut:LREAL;		(* Drehmoment in mNm *)
	tTimeActivOn:TIME;		(* Rampenfunktion Aktiv für FunktionNr 2 --> Zeigt abgelaufene Zeit für die Rampe *)
	tTimeActivOff:TIME;		(* Rampenfunktion Aktiv für FunktionNr 1 --> Zeigt abgelaufene Zeit für die Rampe *)
	rForceCalibrated:REAL;	(* Berechnete Kraft mit Abzug des Kalibrierungswertes *)
	rPosIn:REAL;
END_STRUCT
END_TYPE

(* Data type in Cylinder *)
TYPE ST_CONFIG :
STRUCT
	tDelayOn:TIME;		(* Zeitverzögerung beim einschalten des Zylinders mit der FunktionNr 2-->Timer startet zum Zeitpunkt wenn Ausgang gesetzt wird!
						    Braucht es nur falls die Überwachung des Sensors ausgeschaltet ist-->Nach Ablauf der Zeit wird dann das "xDone-Flag" gesetzt!
						    t=0-->Zeitverzögerung ausgeschaltet *)
	tDelayOff:TIME;		(* Zeitverzögerung beim ausschalten des Zylinders mit der FunktionNr 1-->Timer startet zum Zeitpunkt wenn Ausgang zurück gesetzt wird!
						    Braucht es nur falls die Überwachung des Sensors ausgeschaltet ist-->Nach Ablauf der Zeit wird dann das "xDone-Flag" gesetzt!
						    t=0-->Zeitverzögerung ausgeschaltet *)
	tDelayPreOn:TIME;	(* Zeitverzögerung vor dem einschalten des Zylinders mit der FunktionNr 2-->Nach Ablauf der Zeit wird dann der Ausgang gesetzt,
						    falls nicht auch noch die Zeit "tDelayOn" gesetzt ist!
						    t=0-->Zeitverzögerung ausgeschaltet *)
	tDelayPreOff:TIME;	(* Zeitverzögerung vor dem ausschalten des Zylinders mit der FunktionNr 1-->Nach Ablauf der Zeit wird dann der Ausgang zurück gesetzt,
						    falls nicht auch noch die Zeit "tDelayOff" gesetzt ist!
						    t=0-->Zeitverzögerung ausgeschaltet *)
	xCtrlePosOn:BOOL;	(* FALSE=Sensorüberwachung für FunktionNr 2 ausgeschaltet
						    TRUE=Sensorüberwachung für FunktionNr 2 eingeschaltet-->Mittels der Zeit "tTimeOut" wird festgelegt wie lange auf den Sensor gewartet wird
						     bis ein Fehler generiert wird *)
	xCtrlePosOff:BOOL;	(* FALSE=Sensorüberwachung für FunktionNr 1 ausgeschaltet
						    TRUE=Sensorüberwachung für FunktionNr 1 eingeschaltet-->Mittels der Zeit "tTimeOut" wird festgelegt wie lange auf den Sensor gewartet wird
						     bis ein Fehler generiert wird *)
	tTimeOut:TIME;		(* Gilt für Sensorüberwachung wie lange auf den Sensor gewartet werden muss bis ein Fehler generiert wird *)
	xActivState:BOOL;		(* FALSE=FunktionNr 1 setzt den Ausgang auf TRUE
								  FunktionNr 2 setzt den Ausgang auf FALSE
						    TRUE=FunktionNr 1 setzt den Ausgang auf FALSE
								  FunktionNr 2 setzt den Ausgang auf TRUE *)
END_STRUCT
END_TYPE

(* Data type in Cylinder *)
TYPE ST_CTRLECYL :
STRUCT
(* input *)
	xFBActiv:BOOL;	(* Aktivieren des Zylinder Treiberbausteins *)
	xExecute:BOOL;	(* Ausführen einer Zylinder Funktion *)
	xReset:BOOL;	(* Zurücksetzen des Zylinder Treiberbausteins-->Ausgänge werden auch zurückgesetzt *)
	iFunction:INT;		(*
						1=Zylinder ausschalten-->Grundstellung
						2=Zylinder einschalten
						4=Analogausgang setzen-->Gilt nur für die analogen Zylinderbausteine
						51=Invertieren des Zylinderausganges-->gilt für den Toggle Betrieb
					*)
(* output *)
	xDone:BOOL;			(* Nach dem starten der Funktion wird es zu FALSE und sobald die Funktion beendet wird dann wird es auf TRUE gesetzt!
					    	    sollte ein Fehler entstehen, dann bleibt es auf FALSE bis der Baustein zurückgesetzt wird *)
	xErr:BOOL;			(* Sollte bei einer Funktion ein Fehler entstehen, dann wird dieser Flag gesetzt-->In diesem Fall wird das xDone Flag nicht gesetzt *)
	udiErrorID:UDINT;		(* Fehlernummer, falls des xErr Flag gesetzt wird
							16#F000=Aufgerufene Funktionsnummer gibt es nicht
							16#F201=Bei FunktionNr 2 mit eingeschalteter Sensorüberwachung ist der Sensor nicht eingetroffen-->TimeOut
							16#F202=Bei FunktionNr 1 mit eingeschalteter Sensorüberwachung ist der Sensor nicht eingetroffen-->TimeOut
						*)
	xStatePosOn:BOOL;	(* Sensorzustand für FunktionNr 2 *)
	xStatePosOn1:BOOL;	(* Sensorzustand für FunktionNr 2 -->Falls zweiten Sensor vorhanden ist *)
	xStatePosOff:BOOL;	(* Sensorzustand für FunktionNr 1 *)
	T_Standard:ST_STANDARD;			(* Datenstruktur für Zylinder mit 1 oder 2 Digitalen Ausgänge *)
	T_Analog:ST_ANALOG;				(* Datenstruktur für Zylinder mit nur einem Servoventil *)
END_STRUCT
END_TYPE

(* Data type in Cylinder *)
TYPE ST_CYLINDER :
STRUCT
	iCylinderTpye:INT:=0;		(* 1=CylToolDeflection, 2=CylToolTorque
							     Kann Applikationsbedingt spezifiziert werden *)
	T_Config:ST_CONFIG;		(* Datenstruktur für Grundfunktion aller Zylinder Treiber *)
	T_CtrleCyl:ST_CTRLECYL;	(* Datenstruktur für das Controlling der Zylinder *)
END_STRUCT
END_TYPE

(* Data type in Cylinder *)
TYPE ST_CYLSTAT :  (*Cylinder Status structure to HMI*)
STRUCT
	xOn				:BOOL;
	xOff				:BOOL;
	bStat			:BYTE;
END_STRUCT
END_TYPE

(* Data type in Cylinder *)
TYPE ST_STANDARD :
STRUCT
(* Input *)
	tDelayActiv:TIME;			(* Für die FunktionNr 2 lässt sich mittels dieser Zeit(falls <> 0s) die Impulsdauer festlegen, d.h. der Ausgang bleibt für diese Zeit gesetzt *)
	tDelayAfterSensorOn:TIME;	(* Für die FunktionNr 2 lässt sich mit Sensorüberwachung eine Zeit definieren welches nachdem der Sensor eintrifft bis das Flag xDone gesetzt wird *)
	tDelayAfterSensorOff:TIME;	(* Für die FunktionNr 1 lässt sich mit Sensorüberwachung eine Zeit definieren welches nachdem der Sensor eintrifft bis das Flag xDone gesetzt wird *)
(* Output *)
	xActivOn:BOOL;			(* TRUE falls Ausgang gesetzt ist, anderenfalls FALSE *)
	xActivOff:BOOL;			(* TRUE falls Ausgang für Grundstellung gesetzt ist, anderenfalls FALSE
							     --> Gilt nur für Zylinder mit zwei Ausgänge *)
END_STRUCT
END_TYPE

(* Data type in HDD *)
TYPE ST_CTRLE_HDD :
STRUCT
(* input *)
	xExecute:BOOL:=FALSE;
	xReset:BOOL:=FALSE;
	iFunction:INT:=0;
	tTimeOut:TIME;
	xLocked:BOOL:=FALSE;

(* output *)
	xDone:BOOL:=FALSE;
	xErr:BOOL:=FALSE;
	udiErrorID:UDINT:=0;
END_STRUCT
END_TYPE

(* Data type in HDD *)
TYPE ST_HDD :
STRUCT
	T_Ctrle:ST_CTRLE_HDD;
	T_Config:ST_HDD_CONFIG;
	T_File:ST_HDD_FILE;
	T_Data:ST_HDD_DATA;
END_STRUCT
END_TYPE

(* Data type in HDD *)
TYPE ST_HDD_CONFIG :
STRUCT
	sNetId:T_AmsNetId;
END_STRUCT
END_TYPE

(* Data type in HDD *)
TYPE ST_HDD_DATA :
STRUCT
	sData: ARRAY[1..csiMaxFileLine] OF STRING(csiMaxCharPerLine);
END_STRUCT
END_TYPE

(* Data type in HDD *)
TYPE ST_HDD_FILE :
STRUCT
	sPathAndFileName:STRING(255):='';
	sOldPathAndFileName:STRING(255):='';
	dwPtrWriteBuffer:DWORD:=0;
	udiLenBuffer:UDINT:=0;
	sDirectoryPath:STRING(255):='';
	cssRootPLC:STRING(255):='';
END_STRUCT
END_TYPE

(* Data type in Panel *)
TYPE ST_CTRLEPANEL :
STRUCT
(* Input *)
	xExecute:BOOL:=FALSE;
	iFunction:INT:=0;
	xReset:BOOL:=FALSE;
(* output *)
	xDone:BOOL;
	xErr:BOOL;
	udiErrorID:UDINT;
	udiButton:UDINT:=0;
	udiLED:UDINT:=0;
END_STRUCT
END_TYPE

(* Data type in PASSWORD *)
TYPE ST_PASSWORD :
STRUCT
	T_Ctrle:ST_PASSWORD_CTRLE;
END_STRUCT
END_TYPE

(* Data type in PASSWORD *)
TYPE ST_PASSWORD_CTRLE :
STRUCT
(* input *)
	xExecute:BOOL:=FALSE;
	xReset:BOOL:=FALSE;
	iFunction:INT:=0;
	sGetOperatorPassword : STRING;
	udiGetOperatorPassword : UDINT;
	udiSetOperatorPassword : UDINT;

(* Output *)
	xDone:BOOL:=FALSE;
	xErr:BOOL:=FALSE;
	udiErrorID:UDINT:=0;
END_STRUCT
END_TYPE

(* Data type in PROCESS *)
TYPE ST_CTRLE_PROCESS :
STRUCT
	iFunctNr : INT :=0;
	xEnable : BOOL := FALSE;
	xExecute : BOOL := FALSE;
	xDone : BOOL := FALSE;
	xStop : BOOL := FALSE;
	xRdy : BOOL := FALSE;
	xError : BOOL := FALSE;
	diErrorNr : DINT :=0;
	xErrorReady:BOOL;
	xQuitError : BOOL := FALSE;
	wStatus : WORD := 0;
	xAbordProcess : BOOL := FALSE;
	xReferenced : BOOL := FALSE;
	xActiveProcessState:BOOL:=FALSE;	(* Prozesszustand *)
END_STRUCT
END_TYPE

(* Data type in PROCESS *)
TYPE ST_FCT_PROCESS :
STRUCT
	iFunctNr : INT :=0;
	xExecute: BOOL := FALSE;
	xStop: BOOL := FALSE;
	xQuitError : BOOL := FALSE;
	xAbordProcess : BOOL := FALSE;
	xDone : BOOL := FALSE;
	xError : BOOL := FALSE;
	diErrorNr : DINT := 0;
	xErrorReady:BOOL;
	xSetEndFunction:BOOL;
	xReset:BOOL;
END_STRUCT
END_TYPE

(* Data type in PROCESS *)
TYPE ST_PREWARNING :
STRUCT
	xToolNearChangeSt1:BOOL;			(* Dieses Signal besagt dass bald ein Werkzeug Wechsel vorgenommen werden muss *)
	xZAxisBrakeBlockedSt1:BOOL;		(* Dieses Signal besagt dass die Bremse der Z Achse blockiert ist *)

	asMessageBufferEngl:ARRAY [1..10,1..5] OF STRING(55);	(* Maximal 10 Meldungen können aufgenommen werden *)
	asMessageBufferGer:ARRAY [1..10,1..5] OF STRING(55);	(* Maximal 10 Meldungen können aufgenommen werden *)

	aiMessageNrBuffer:ARRAY [1..10] OF INT;			(* Maximal 10 Meldungen-->Nummer der Meldung *)
	xPreWarningActive:BOOL;							(* Dieses Signal besagt ob mindestens eine Vorwarnung besteht *)
	iNumberOfMessage:INT;								(* Anzahl eingetragenen Meldungen *)
	asEmptyMessageEngl:ARRAY [1..5] OF STRING(55);		(* Diese Meldung wird angezeigt wenn keine Warnungen vorhanden sind *)
	asEmptyMessageGer:ARRAY [1..5] OF STRING(55);		(* Diese Meldung wird angezeigt wenn keine Warnungen vorhanden sind *)
	aiDeleteMessage:ARRAY [1..10] OF INT;				(* Nummer zu löschende Meldung *)
END_STRUCT
END_TYPE

(* Data type in PROCESS *)
TYPE ST_PROCESS :
STRUCT
	T_Ctrle:ST_CTRLE_PROCESS;
	T_Fct:ST_FCT_PROCESS;
END_STRUCT
END_TYPE

(* Data type in ProcessData *)
TYPE ST_PROCESSDATA :
STRUCT
	T_Ctrle:ST_PROCESSDATA_CTRLE;
END_STRUCT
END_TYPE

(* Data type in ProcessData *)
TYPE ST_PROCESSDATA_CTRLE :
STRUCT
(* input *)
	xExecute:BOOL:=FALSE;
	xReset:BOOL:=FALSE;
	iFunction:INT:=0;
(* Output *)
	xDone:BOOL:=FALSE;
	xErr:BOOL:=FALSE;
	udiErrorID:UDINT:=0;
	tTimeElapsed:TIME;
END_STRUCT
END_TYPE

(* Data type in Profile *)
TYPE ST_PROFILE :
STRUCT
	T_Ctrle:ST_PROFILE_CTRLE;
	T_Id:ST_PROFILE_ID;
	T_LoadProfileParameter:ST_RETAIN_DATA_PROFILEPARAMETER;	(* Profil Parameter für Profil(LoadData) *)
	T_ProcProfileParameter:ST_RETAIN_DATA_PROFILEPARAMETER;	(* Prozessabblid Parameter für Profil(Data) *)
	T_DefaultProfileParameter:ST_RETAIN_DATA_PROFILEPARAMETER;	(* Default Werte für OnlineChange und Prozess Parameter *)
	T_CopyProfileParameter:ST_RETAIN_DATA_PROFILEPARAMETER;					(* Braucht es nur damit die eingelesenen Werte eines Profils kopiert werden können *)
	T_Profile_MinMax:ST_PROFILEONLINECHANGE;
	T_IDProfileStation:ARRAY[1..csiMaxProfile] OF ST_PROFILE_ID;
END_STRUCT
END_TYPE

(* Data type in Profile *)
TYPE ST_PROFILE_CTRLE :
STRUCT
(* input *)
	xExecute:BOOL:=FALSE;
	xReset:BOOL:=FALSE;
	iFunction:INT:=0;
	sPathAndFileName:STRING(255):='';
	sProfileName:STRING(30);
	xActiveReadProfileForCopy:BOOL;

(* Output *)
	xDone:BOOL:=FALSE;
	xErr:BOOL:=FALSE;
	udiErrorID:UDINT:=0;
END_STRUCT
END_TYPE

(* Data type in Profile *)
TYPE ST_PROFILE_ID :
STRUCT
	iNumber:INT;
	sName:STRING(30);
END_STRUCT
END_TYPE

(* Data type in Profile *)
TYPE ST_PROFILE_LIST :
STRUCT
	iNumber:INT;
	sName:STRING(30);
END_STRUCT
END_TYPE

(* Data type in Profile *)
TYPE ST_PROFILE_LIST_MANAGE :
STRUCT
	xListProfileUp:BOOL;
	xListProfileDown:BOOL;
END_STRUCT
END_TYPE

(* Data type in Profile *)
TYPE ST_PROFILEONLINECHANGE :
STRUCT
	T_Max:ST_PROFILEONLINECHANGE_DATA;
	T_Min:ST_PROFILEONLINECHANGE_DATA;
END_STRUCT
END_TYPE

(* Data type in Profile *)
TYPE ST_PROFILEONLINECHANGE_DATA :
STRUCT
	rTorqueLevelHC:REAL;								(* Schwellwert Drehmoment HC-->Gleichwertig wie konventionell ein HC ausgelöst wurde *)
	rForceDeflection:REAL;
	rWorkingSpeedForward:REAL;						(* Normalgeschwindigkeit ohne dass Schwellwert Drehoment Aktiv ist *)
	rWorkingOffsetBackward:REAL;
	rWorkingSpeedBackward:REAL;
	rWorkingSpindleSpeed:REAL;
END_STRUCT
END_TYPE

(* Data type in Retain *)
TYPE ST_CTRLE_DATA_RETAIN :
STRUCT
(* input *)
	xExecute:BOOL:=FALSE;
	xReset:BOOL:=FALSE;
	iFunction:INT:=0;
	udiSrcLen:UDINT;
	udiDestLen:UDINT;
	udipSrcAddr:UDINT;
	udipDestAddr:UDINT;
	tTimeOut:TIME;
	xBlockReadFirstTime:BOOL;

(* Output *)
	xFirstRead:BOOL:=FALSE;
	xDone:BOOL:=FALSE;
	xErr:BOOL:=FALSE;
	udiErrorID:UDINT:=0;
END_STRUCT
END_TYPE

(* Data type in Retain *)
TYPE ST_NOVRAM :
STRUCT
	T_Ctrle:ST_CTRLE_DATA_RETAIN;
	T_Parameter:ST_RETAIN_DATA;
END_STRUCT
END_TYPE

(* Data type in Retain *)
TYPE ST_RETAIN_DATA :
STRUCT
	T_Machine:ST_RETAIN_DATA_MACHINE;
	T_StationWork: ARRAY [1..1] OF ST_RETAIN_DATA_STATIONWORK;
	T_ErrorNrList:ST_RETAIN_ERROR_DATA;
	T_PartAnalysis:ARRAY [1..1] OF ST_PARTANALYSIS;

	arZ1AxisCalcEndPosSaveProfile:ARRAY [1..1,1..100] OF REAL;	(* Zu jedem Profil wird die Endposition für das Inkrementieren der Z EndPos gespeichert. So hat man die Möglichkeit wenn man das Profil ändert und dann wieder ein bestehendes Profil wieder laded und immer noch mit dem
															   gleichen Wz arbeitet, dass dieser Wert immer noch vorhanden ist. Wenn man aber für dieses Profil ein neues Wz einspannt, dann muss der Bediener den Zählerstand nullen, anderenfalls fährt es dann tiefer *)

	arZ1CentringCalcEndPosSaveProfile:ARRAY [1..1,1..100] OF REAL;	(* Zu jedem Profil wird die Endposition für das Inkrementieren der Z Zentrierpos gespeichert. So hat man die Möglichkeit wenn man das Profil ändert und dann wieder ein bestehendes Profil wieder laded und immer noch mit dem
															   gleichen Wz arbeitet, dass dieser Wert immer noch vorhanden ist. Wenn man aber für dieses Profil ein neues Wz einspannt, dann muss der Bediener den Zählerstand nullen, anderenfalls fährt es dann tiefer *)
END_STRUCT
END_TYPE

(* Data type in Retain *)
TYPE ST_RETAIN_DATA_AX5000_PARAM :
STRUCT
	uiP61					: UINT;								(* Parameter P-0-0061 *)
	bP150					: ARRAY [0..227] OF BYTE;				(* Parameter P-0-0150 *)
END_STRUCT
END_TYPE

(* Data type in Retain *)
TYPE ST_RETAIN_DATA_MACHINE :
STRUCT
	T_ParamSystem:ST_EXCHG_PARAM_SYSTEM;
	T_ParamAutomat:ST_EXCHG_PARAM_AUTOMAT;
	adiPotentiometerValue		:ARRAY [0..11] OF DINT;	(* Wert für Potentiometerstellung *)
	xEndlessProcessActive:BOOL;
END_STRUCT
END_TYPE

(* Data type in Retain *)
TYPE ST_RETAIN_DATA_PROFILEPARAMETER :
STRUCT
	T_ProzessData:ST_EXCHG_PARAM_STANDARDPROCESS;
	T_ProfileOnlineChange:ST_PROFILEONLINECHANGE_DATA;
END_STRUCT
END_TYPE

(* Data type in Retain *)
TYPE ST_RETAIN_DATA_STATIONWORK :
STRUCT
	T_StProcess:ST_EXCHG_PARAM_STANDARDPROCESS;	(* Standard Parameter Prozessabbild ohne dass das Profile geändert wird-->Prozess arbeitet mit diesen Parameter *)
	T_OnlineChange:ST_PROFILEONLINECHANGE_DATA;	(* OnlineChange Parameter Prozessabbild ohne dass das Profile geändert wird-->Prozess arbeitet mit diesen Parameter *)
	T_OnlineChangeINC:ST_PROFILEONLINECHANGE_DATA;
	T_InfoProcess:ST_EXCHG_INFO_PROCESS;
	T_AxisState:ST_EXCHG_PARAM_AXIS_STATE;
	T_TorqueSystem:ST_EXCHG_PARAM_TORQUESYSTEM;					(* Maxon Spindel *)
	T_TorqueSystem_L:ST_EXCHG_PARAM_TORQUESYSTEM_L;				(* Beckhoff Spindel L *)
	T_TorqueSystem_M:ST_EXCHG_PARAM_TORQUESYSTEM_L;				(* Beckhoff Spindel M *)		(* IGS *)
	T_SpindleSystem:ST_EXCHG_PARAM_SPINDLESYSTEM;					(* Maxon Spindel *)
	T_SpindleSystem_L:ST_EXCHG_PARAM_SPINDLESYSTEM_L;				(* Beckhoff Spindel L *)
	T_SpindleSystem_M:ST_EXCHG_PARAM_SPINDLESYSTEM_L;				(* Beckhoff Spindel M *)		(* IGS *)
	T_Fct_SpindleBurnIn:ST_EXCHG_PARAM_SPINDLEBURNIN;
	T_Fct_SpindleCalibration:ST_EXCHG_PARAM_SPINDLECALIBRATION;
	T_ToolCounter:ST_EXCHG_PARAM_TOOLCOUNTER;
	T_WPCounter:ST_EXCHG_PARAM_WPCOUNTER;
	(* Zylinder Parameter für WorkStation MicroHead *)
	TCylBrakeReleaseZAxis:ST_EXCHG_PARAM_CYLINDER;
(* Gilt für das Aufzeichnen der Rotationsdauer der Spindel *)
	tSpindelActiveRotationTime:TIME;
	iSpindelActiveRotationDay:INT;
	tSpindel2ActiveRotationTime:TIME;										(* IGS *)
	iSpindel2ActiveRotationDay:INT;										(* IGS *)
	tSpindel3ActiveRotationTime:TIME;										(* IGS *)
	iSpindel3ActiveRotationDay:INT;										(* IGS *)
	T_RegulatorSpindle_SM:ST_EXCHG_PARAM_CONTRMOT;
	T_Z_TGuide:ST_EXCHG_PARAM_Z_TGUIDE;

	T_AxisS2:ST_RETAIN_DATA_AX5000_PARAM;	(* AX5000 Parameter *)		(* Beckhoff Spindel L *)		(* IGS *)
	T_AxisS3:ST_RETAIN_DATA_AX5000_PARAM;	(* AX5000 Parameter *)		(* Beckhoff Spindel M *)		(* IGS *)
END_STRUCT
END_TYPE

(* Data type in Retain *)
TYPE ST_RETAIN_ERROR_DATA :
STRUCT
	adiErrorListMachine:ARRAY [1..20] OF DINT;
	asErrorTimeStampMachine:ARRAY [1..20] OF STRING(12);
END_STRUCT
END_TYPE

(* Data type in StartUp *)
TYPE ST_CTRLESTARTUP :
STRUCT
(* Input *)
	xExecute:BOOL;
	xReset:BOOL;
	iFunction:INT;
	iMsgNumber:INT;
	xUnlockSecurityDoor:BOOL;
	xSetSecurityStateON:BOOL;
	xDeleteAllMessageOverlay:BOOL;
(* Output *)
	xDone:BOOL;
	xErr:BOOL;
	udiErrorID:UDINT;
END_STRUCT
END_TYPE

(* Data type in StartUp *)
TYPE ST_STARTUP :
STRUCT
	T_Ctrle:ST_CTRLESTARTUP;
	T_State:ST_STARTUPSTATE;
END_STRUCT
END_TYPE

(* Data type in StartUp *)
TYPE ST_STARTUPSTATE :
STRUCT
	xPLCReady:BOOL;
	xCompleted:BOOL;
	xBlockChangeMovementVisu:BOOL;
END_STRUCT
END_TYPE

(* Data type in STATIC_ERROR_LIST *)
TYPE ST_ERROR_LIST :
STRUCT
	asErrorListEnglish: ST_LANGUAGE_LIST;
	asErrorListDeutsch: ST_LANGUAGE_LIST;
	asErrorListFrancais: ST_LANGUAGE_LIST;
END_STRUCT
END_TYPE

(* Data type in STATIC_ERROR_LIST *)
TYPE ST_LANGUAGE_LIST :
STRUCT
	T_LanguagList:ARRAY [1..300] OF STRING(100);
END_STRUCT
END_TYPE

(* Data type in StationsControlling/PART_ANALYSIS *)
TYPE ST_PARTANALYSIS :
STRUCT
	sFileName:STRING;
	sStartOfProcess:STRING;
	sEndOfProcess:STRING;
	diActual_NumberHoleToWork:DINT;					(* Aktuell zu bearbeitende Bohrungsnummer *)

	abWorkPartQuality:ARRAY [1..ciMaxWP] OF BYTE;		(* 0=Hole not worked, 1=Go HC, 2=Go No HC, 3=NoGo minTime, 4=NoGo maxTime, 5=NoGo insert fail, 6=NoGo NoWP detect, 7=Working, 8=Cycle aborted *)
	arFirstHC:ARRAY [1..ciMaxWP] OF REAL;				(* Absolute Position der Z-Achse in mm beim ersten HC *)
	aiHCCounter:ARRAY [1..ciMaxWP] OF INT;			(* Anzahl HC *)
	aiHCCounterCentering:ARRAY [1..ciMaxWP] OF INT;			(* Anzahl HC während der Zentrierung *)
	aiHCCounterTorque:ARRAY [1..ciMaxWP] OF INT;		(* Anzahl HC *)
	aiHCCounterSpeed:ARRAY [1..ciMaxWP] OF INT;		(* Anzahl HC Geschwindigkeit *)		(* IGS *)
	adiCycleTime:ARRAY [1..ciMaxWP] OF DINT;			(* Zykluszeit in ms --> Beinhaltet Wstk Spannung, Spindeldrehung, Bearbeitung, Spindel stoppen und Wstk entspannen *)
	adiWorkTime:ARRAY [1..ciMaxWP] OF DINT;			(* Bearbeitungszeit --> Beinhaltet nur die effektive Bearbeitungszeit *)
	abInfeedCounterZ:ARRAY [1..ciMaxWP] OF BYTE;		(* Anzahl Einfädelversuche mit der Z Achse. Wenn erste mal durchgeht dann steht eine 1, wenn erst beim zweiten Versuch dann eine 2 usw. *)
	adiNumberHole:ARRAY [1..ciMaxWP] OF DINT;		(* WstkNummer *)
END_STRUCT
END_TYPE

(* Data type in StationsControlling/PART_ANALYSIS *)
TYPE ST_PARTANALYSIS_OUTPUT :
STRUCT
	bHole_WorkPartQuality:BYTE;		(* 0=Hole not worked, 1=Go HC, 2=Go No HC, 3=NoGo minTime, 4=NoGo maxTime, 5=NoGo insert fail, 6=NoGo NoHole, 7=Working, 8=Cycle aborted *)
	rHole_FirstHC:REAL;				(* Absolute Position der Z-Achse in mm beim ersten HC *)
	iHole_HCCounter:INT;				(* Anzahl HC Deflection *)
	iHole_HCCounterCentering:INT;		(* Anzahl HC Deflection beim Zentrieren *)
	iHole_HCCounterTorque:INT;		(* Anzahl HC Drehmoment *)
	iHole_HCCounterSpeed:INT;		(* Anzahl HC Z Geschwindigkeit *)	(* IGS *)
	diHole_CycleTime:DINT;			(* Zykluszeit in ms --> Beinhaltet Wstk Spannung, Spindeldrehung, Bearbeitung, Spindel stoppen und Wstk entspannen *)
	diHole_WorkTime:DINT;			(* Bearbeitungszeit --> Beinhaltet nur die effektive Bearbeitungszeit *)
	bHole_InfeedCounterZ:BYTE;		(* Anzahl Einfädelversuche mit der Z Achse. Wenn erste mal durchgeht dann steht eine 1, wenn erst beim zweiten Versuch dann eine 2 usw. *)
	diHoleNumber:DINT;
END_STRUCT
END_TYPE

(* Data type in StationsControlling/STATION_WORK *)
TYPE ST_CTRL_ONLINECHANGE :
STRUCT
(* Online Change Synch *)
	xLockChange_Z_WorkSpeedForward:BOOL:=TRUE;
	xLockChange_Z_WorkSpeedBackward:BOOL:=TRUE;
	xLockChange_S_WorkSpindleSpeed:BOOL:=TRUE;
	xLockChangeCylToolTorqueLevel:BOOL:=TRUE;
	xLockChangeCylToolDeflectionForce:BOOL:=TRUE;
END_STRUCT
END_TYPE

(* Data type in StationsControlling/STATION_WORK *)
TYPE ST_CTRL_WORK :
STRUCT
	rLastOverLimitPosition:REAL:=0.0;
	iOverLimitCounter:INT:=0;
	iOverLimitCounterCentering:INT:=0;
	iOverLimitCounterTorque:INT:=0;
	iOverLimitCounterSpeed:INT:=0;				(* IGS *)
	rDiffOverLimitPosition:REAL:=0.0;
	rActualFirstContactPosition:REAL:=0.0;
	rLastFirstContactPosition:REAL:=0.0;
	bPartQuality:BYTE; 	(* 0=Hole not worked, 1=Go HC, 2=Go No HC, 3=NoGo minTime, 4=NoGo maxTime, 5=NoGo insert fail, 6=NoGo NoWP detect, 7=Working, 8=Cycle aborted, 9=No WP, 10=NoGo HC Centr., 11=WP Centered *)
	rEffCycleTime : REAL;	(* Effektive Bearbeitungszeit-->Timer startet nach dem ersten Ausschlag-->sollte kein Ausschlag eintreffen dann ist diese Zeit = 0 *)
	rCuttingSpeed:REAL;	(* Schnittgeschwindigkeit *)

(* Drehmoment Ausgabe für den Prozess in Abhängigkeit der HubAchsen Position *)
	xActiveProcess_CylToolTorqueHC:BOOL;
	xBlockOutput_CylToolTorqueHC:BOOL;

	rTorqueHC:REAL;
	rTorqueAfterHC_Min:REAL;
	rTorqueAfterHC_Max:REAL;
	xTorqueLastHC:BOOL;
	xDeflectionLastHC:BOOL;
	iHCTorquePos:INT;
	iHCDeflectionPos:INT;
	xHCSparkOut:BOOL;

(* Regler *)
	rSpeedZ_V1:REAL;						(* IGS *)
	rSpeedZ_V3:REAL;						(* IGS *)
	rTorqueZ_S1:REAL;						(* IGS *)
	rTorqueZ_S4:REAL;						(* IGS *)
	iProgressBar_Torque:INT;					(* IGS *)
	iProgressBar_ZPos:INT;					(* IGS *)
	iProgressBar_ZVel:INT;					(* IGS *)
	xTorqueAfterHC_Min_Overlimit:BOOL;		(* IGS *)
	xTorqueAfterHC_Max_Overlimit:BOOL;		(* IGS *)

	xDoNotMoveZPosition:BOOL;

	xActiveProcess:BOOL;				(* Gilt nur für das Kühlmittel *)
	xStationBlocked:BOOL;				(* Gilt für die Werkzeugspannung, als Sicherheit für den Teller *)
	iStationBlockedErrNr:INT;			(* Gilt für die Werkzeugspannung, als Sicherheit für den Teller, welcher Aktuator aktiv ist *)
	xWorkingFinished:BOOL;
	xWorkingStarted:BOOL;

	xWorkStartToolRotation:BOOL;
	xWorkStopToolRotation:BOOL;

	rMaxToolSpindleSpeed:REAL;

	xStopToolRotation:BOOL;

(* Gilt für die Kalibrierungsporzedur-->mittels diesen Flag kann mittgeteilt werden ob ToolDeflection und/oder ToolTorque kalibriert werden muss *)
	xActiveCalibrateToolDeflection:BOOL;
	xActiveCalibrateToolTorque: BOOL;	(*  *)
	rOffsetToolDeflection:REAL;
	rOffsetToolTorque:REAL;

(* Gilt für das Aufzeichnen der Rotationsdauer der Spindel *)
	tSpindelActiveRotationTime:TIME;
	iSpindelActiveRotationDay:INT;
	tSpindel2ActiveRotationTime:TIME;			(* IGS *)
	iSpindel2ActiveRotationDay:INT;			(* IGS *)
	tSpindel3ActiveRotationTime:TIME;			(* IGS *)
	iSpindel3ActiveRotationDay:INT;			(* IGS *)

(* Gilt für die Ausfunkprozedur bezüglich der Kraftmessdose für das Drehmoment *)
	xSparkOutActive:BOOL;
(* Gilt für die Erstinitialisierung der Z Achse *)
	iInitialMode_Z_Axis:INT;
	lrSaveTeachedPosition:LREAL;

(* Ausgabe für Wstk Zähler Maschine und Stationen *)
	xAddWPCounter_Machine_IO:BOOL;		(* Inkrementiere Maschinen WstkZähler für IO Wstk *)
	xAddWPCounter_Machine_NIO:BOOL;	(* Inkrementiere Maschinen WstkZähler für NIO Wstk *)
	xAddToolCounter_Machine:BOOL;		(* Inkrementieren bearbeitete Bohrungen für den WzZähler *)

	xToolInfeeded:BOOL;	(* Besagt ob das Wz eingefädelt werden konnte *)

	xWP_Analyse_ActiveCycle:BOOL;			(* Zykluszeit für zu bearbeitende Bohrung ist gestartet *)
	xWP_Analyse_ActiveWork:BOOL;			(* Bearbeitungszeit für zu bearbeitende Bohrung ist gestartet *)
	xWP_Analyse_ReadyToReadData:BOOL;	(* Gilt für das Synchronisieren der Daten für die Wstk Daten Analyse *)
	xWP_Analyse_StartAutomat:BOOL;			(* Gilt für die Aufzeichnungsdatei, um festzulegen wann der Automat für das jeweilige Talon gestartet wurde *)
	xWP_Analyse_StopAutomat:BOOL;			(* Gilt für die Aufzeichnungsdatei, um festzulegen wann der Automat für das jeweilige Talon beendet wurde *)

	xLastTryInfeed:BOOL;

(* Gilt für die Blockierung der Achsenbremse *)
	xZAxisBrakeBlocked:BOOL;
	xBlockCheckAxisBrake:BOOL;

	rProcessWork:REAL;						(* Bearbeitungsarbeit *)		(* IGS *)
END_STRUCT
END_TYPE

(* Data type in StationsControlling/STATION_WORK *)
TYPE ST_HW_WORKSTATION :
STRUCT
	xActiveStation:BOOL;
	TCtrlWork 						:ST_CTRL_WORK;

	TAxisZ 							:ST_AXIS;			(* Achse für die Hubachse Z *)
	TAxisS 							:ST_AXIS;			(* Achse für die Werkzeugspindel *)
	TCylToolDeflection				:ST_CYLINDER;		(* Servoventil für das bestimmen der vertikalen Auslenkraft für SM oder L Spindelkopf *)
	TCylToolTorqueHC 				:ST_CYLINDER;		(* Servoventil für Drehmomentüberwachung HC für SM oder L Spindelkopf *)
	TCylToolTorqueOverload 			:ST_CYLINDER;		(* Servoventil für Drehmomentüberwachung Überlast für SM oder L Spindelkopf *)
	TSensorTorque 					:ST_CYLINDER;		(* Analoger Sensor für Drehmoment detektion *)
	TSensorTorqueOverload 			:ST_CYLINDER;		(* Digitaler Sensor für Drehmoment Überlast detektion *)										(* IGS *)
	TTorqueSensorMeasRange		:ST_CYLINDER;		(* Controlling für den Drehmomentsensor, Einstellung des Drehmomentbereiches *)				(* IGS *)
	TTorqueSensorControl				:ST_CYLINDER;		(* Controlling für den Drehmomentsensor, Überprüfung auf Funktionalität *)						(* IGS *)
	TSensorToolSpindle_L_Connect 	:ST_CYLINDER;		(* Digitaler Sensor für Spindelkopf L angeschlossen *)
	TCylBrakeReleaseZAxis 			:ST_CYLINDER;		(* Zylinder für lösen der Bremse bei der Z Achse *)
	TCylWorkpieceClamp				:ST_CYLINDER;		(* Ventil für Werkstückfixierzylinder *)
	TValveAirTable					:ST_CYLINDER;		(* Ventil für die Luft des Tisches *)
	TValveVacuumTable				:ST_CYLINDER;		(* Ventil für die Luft des Tisches *)
	TAxisBubbler						:ST_DC_AXIS;		(* Rührwerk für Suspension *)															(* IGS3 *)
	TAxisFeedPump					:ST_DC_AXIS;		(* Förderpumpe für Suspension *)														(* IGS3 *)
END_STRUCT
END_TYPE

(* Data type in StationsControlling *)
TYPE ST_CTRLE_STATION :
STRUCT
	xActiveStation : BOOL;
	xActiveHardware : BOOL;
	xHardwareConfigError : BOOL;
	iFunctNr : INT :=0;
	xEnable : BOOL := FALSE;
	xSecurityCircuitOn : BOOL := FALSE;
	xSecurityCircuitOff : BOOL := FALSE;
	xExecute : BOOL := FALSE;
	xDone : BOOL := FALSE;
	xStop : BOOL := FALSE;
	xStopCycle : BOOL :=FALSE;
	xRdy : BOOL := FALSE;
	xError : BOOL := FALSE;
	diErrorNr : DINT :=0;
	xQuitError : BOOL := FALSE;
	wStatus : WORD := 0;
	xAbord : BOOL := FALSE;
	xReferenced : BOOL := FALSE;
	xResetReference : BOOL :=FALSE;
	xSetReference : BOOL :=FALSE;
	xHWAxesActive : BOOL := FALSE;
	xActiveMovement : BOOL;
	xResetHardware:BOOL;
	xResetHardwareActivateCurrent:BOOL;
	xSaveParameterToNovRAM:BOOL;
	xBlockCheckZylinder:BOOL;
END_STRUCT
END_TYPE

(* Data type in StationsControlling *)
TYPE ST_STATION :
STRUCT
(* Controlling *)
	xActive : BOOL;
	iStationNr:INT;
	sStationName : STRING(30);
(* Layer 3 *)
	TControl : ST_CTRLE_STATION;
	TCtrlOnlineChange:ST_CTRL_ONLINECHANGE;
(* Layer 2 *)
	THWWorkStation 		:ST_HW_WORKSTATION;
END_STRUCT
END_TYPE

(* Data type in Terminals *)
TYPE ST_TERMINAL_STATE :
STRUCT
	wEtherCAT_1_State:WORD;				(* 0 =No Error *)
	wEtherCAT_2_State:WORD;				(* 0 =No Error *)
	wWCMasterAxisModul1_State:WORD;		(* 8 =Operational Mode (OP) *)
	wWCMasterAxisModul2_State:WORD;		(* 8 =Operational Mode (OP) *)
	wWCEPOS_State:WORD;					(* 8 =Operational Mode (OP) *)
	wWCSMCValve:WORD;					(* 8 =Operational Mode (OP) *)
END_STRUCT
END_TYPE

(* Data type in TwinSAFE *)
TYPE ST_SAFETY_STATUS :
STRUCT
(*Status, dependent to the Safety-Program, for use in PLC*)
	iSetupMode							:INT;(*1=Mode'A', 2=Mode'B', 0=NormalBetrieb'*)

	xSetupOperateModeActive			:BOOL;

	xEnergyONNormalMode				:BOOL;

	xEnergyONSetupModeASt1			:BOOL;

	xEnergyONSetupModeBSt1			:BOOL;

	xMachineDoorClose					:BOOL;

	xMachineEmergStopActive			:BOOL;

	xSecuritySwitch						:BOOL;
	xSecurityDoorOpen					:BOOL;		(* Maschinentüre und/oder Ladetüre offen *)
	xSecurityDoorClose					:BOOL;		(* Maschinentüre und Ladetüre geschlossen *)
END_STRUCT
END_TYPE

(* Data type in TwinSAFE *)
TYPE ST_TWINSAFE_CTRLE_IN :
STRUCT
	xTwinSAFE_Group_FB_Error_1: BOOL;
	xTwinSAFE_Group_COM_Error_1: BOOL;
	xTwinSAFE_Group_OUT_Error_1: BOOL;
END_STRUCT
END_TYPE

(* Data type in TwinSAFE *)
TYPE ST_TWINSAFE_CTRLE_OUT :
STRUCT
	xTwinSAFE_Run_1: BOOL;
	xTwinSAFE_Reset_1: BOOL;
END_STRUCT
END_TYPE

(* Data type in TwinSAFE *)
TYPE ST_TWINSAFE_DRIVE :
STRUCT
(* Standard Sicherheitsfunktionen *)
	xSTO: BOOL;		(* Safe Torque Off *)
	xSS1: BOOL;		(* Safe Stop1 *)
	xSS2: BOOL;		(* Safe Stop2 *)
	xSOS: BOOL;		(* Safe Operating Stop *)
	xSSR: BOOL;		(* Safe Speed Range *)
	xSDIp: BOOL;		(*Safe Direction Positive *)
	xSDIn: BOOL;		(* Safe Direction Negative *)
(* Zusätzliche Sicherheitsfunktionen *)
	xSLS1: BOOL;		(* Safe Limited Speed 1 *)
	xSLS2: BOOL;		(* Safe Limited Speed 2 *)
	xSSM: BOOL;		(* Safe Speed Monitor *)
	xSMS: BOOL;		(* Safe Maximum Speed *)
	xSLP: BOOL;		(* Safe Limited Position *)
	xSCA: BOOL;		(* Safe CAM *)
	xSLI: BOOL;		(* Safe Limited Increment *)
	xSAR: BOOL;		(* Safe Acceleration Range *)
	xSMA: BOOL;		(* Safe Maximum Acceleration *)
	xError: BOOL;		(* Errorausgabe oder Error Quittierung *)
END_STRUCT
END_TYPE

(* Data type in TwinSAFE *)
TYPE ST_TWINSAFE_FB_ERROR :
STRUCT
(*Fehlermeldungen der FB's in Safety-PLC*)
	xMON_EmergencyButtonMachine		:BOOL;	(* Diskrepanzfehler  Not Aus Taster Maschine *)
	xMON_Error_MachineDoor				:BOOL;	(* Diskrepanzfehler Sicherheitstüre der Maschine *)
	xMON_KeySwitchProcObservation		:BOOL;	(* Diskrepanzfehler Schlüsselschalter für Einrichtbetrieb Prozessbeobachtung Stellung I *)
	xMON_KeySwitchWorkStation			:BOOL;	(* Diskrepanzfehler Schlüsselschalter für Einrichtbetrieb Bearbeitungsstation Stellung II *)
	xMON_EnablingSwitchActive				:BOOL;	(* Diskrepanzfehler Zustimmschalter *)
	xMON_AxesCurrentOff					:BOOL;	(* Diskrepanzfehler Antriebsperrtaste *)
	xEDM_PowSup_MasterModul			:BOOL;	(* Fehler im Rückführkreis der Leistungsschütze der Z1 Achse (400V) *)
	xEDM_PowSup_24V					:BOOL;	(* Fehler im Rückführkreis des Sicherheitsrelais für 24V Speisung *)
END_STRUCT
END_TYPE

(* Data type in TwinSAFE *)
TYPE ST_TWINSAFE_IN :
STRUCT
(* EL1904, Input *)
	IxEmergencyStopButtonCh1:BOOL;			(* Notaus Taste Kanal 1 *)
	IxEmergencyStopButtonCh2:BOOL;			(* Notaus Taste Kanal 2 *)
	IxKeySwitchProcObservationCh1:BOOL;		(* Schlüsselschalter für Einrichtbetrieb Prozessbeobachtung Kanal 1, Stellung I *)
	IxKeySwitchProcObservationCh2:BOOL;		(* Schlüsselschalter für Einrichtbetrieb Prozessbeobachtung Kanal 2, Stellung I *)
	IxKeySwitchWorkStationCh1:BOOL;			(* Schlüsselschalter für Einrichtbetrieb Bearbeitungsstation Kanal 1, Stellung II *)
	IxKeySwitchWorkStationCh2:BOOL;			(* Schlüsselschalter für Einrichtbetrieb Bearbeitungsstation Kanal 2, Stellung II *)
	IxEnablingSwitchActiveCh1:BOOL;			(* Zustimmschalter, Stellung 2-Aktiv, K1 *)
	IxEnablingSwitchActiveCh2:BOOL;			(* Zustimmschalter, Stellung 2-Aktiv, K2 *)
	IxCabinDoorCloseCh1:BOOL;				(* Kabinentüre Maschine (Sicherheitstüre) geschlossen, Kanal 1 *)
	IxCabinDoorCloseCh2:BOOL;				(* Kabinentüre Maschine (Sicherheitstüre) geschlossen, Kanal 2 *)
	IxCabinDoorOpen:BOOL;					(* Kabinentüre Maschine (Sicherheitstüre) GEöffnet *)
	IxContactorAuxContact24V:BOOL;			(* Rückführkreis des Sicherheitsrelais für 24V Speisung *)
	IxAxesCurrentOffCh1:BOOL;					(* Externe Taste füR das Ausschalten der Achsen Energieversorgung, Kanal 1 *)
	IxAxesCurrentOffCh2:BOOL;					(* Externe Taste füR das Ausschalten der Achsen Energieversorgung, Kanal 2 *)
	IxContactorAuxContactMasterModul:BOOL;	(* Rückführkreis der Leistungsschütze Z1, S (400V) *)
	IxCabinDoorClose:BOOL;					(* Kabinentüre Maschine geschlossen, Näherungsschalter (Induktiv) *)
	IxReadyToOperateMasterModul1:BOOL;		(* Betriebsbereitschaftsausgabe von Z1  Achse (BTB) *)
	IxReadyToOperateMasterModul2:BOOL;		(* Betriebsbereitschaftsausgabe von S Achse (BTB) *)	(* IGS *)
	IxRes19:BOOL;							(* Reserve *)
	IxRes20:BOOL;							(* Reserve *)
END_STRUCT
END_TYPE

(* Data type in TwinSAFE *)
TYPE ST_TWINSAFE_OUT :
STRUCT
(* EL2904, Output *)
	QxContactorMasterModul400VCh1:BOOL;		(* Einschalten der Leistungsschütze  Z1-, S-Achse 400V, Kanal 1 *)
	QxContactorMasterModul400VCh2:BOOL;		(* Einschalten der Leistungsschütze  Z1-, S-Achse 400V, Kanal 2 *)
	QxContactor24VCh1:BOOL;					(* Einschalten des Sicherheitsrelais für 24V Speisung, Kanal 1 *)
	QxContactor24VCh2:BOOL;					(* Einschalten des Sicherheitsrelais für 24V Speisung, Kanal 2 *)
	QxEnablingAxisSpindle_St1:BOOL;			(* Freigabe Spindel Arbeitsstation *)
	QxEnablingSwitchLed:BOOL;				(* Zustimmschalter Bereitschaftsanzeige *)
	QxRes56:BOOL;							(* Reserve *)
	QxRes57:BOOL;							(* Reserve *)
END_STRUCT
END_TYPE

(* Data type in UPS *)
TYPE ST_CTRLE_UPS :
STRUCT
(* input variable *)
	xDIPDisable:BOOL:=TRUE;
	iDischargeLevel : USINT:=2;
	tDelay:TIME:=T#3s;
(* output variable *)
	xPowerFailure:BOOL;
	xShutdownActive:BOOL;
	xUPSReady:BOOL;
	x24VInOK:BOOL;
	xHolding:BOOL;
	tTimeUntilShutdown:TIME;
	eUPSState : E_UPS_STATE;
	xBlockSystem_PowerFail:BOOL;
END_STRUCT
END_TYPE

(* Data type in VISUALISIERUNG *)
TYPE ST_BUTTON :
STRUCT
	xInputState:BOOL;
	xLedState:BOOL;
	xResetTime:BOOL;
	tPressTime:TIME;
END_STRUCT
END_TYPE

(* Data type in VISUALISIERUNG *)
TYPE ST_CONFIGPAGE :
STRUCT
	sName:STRING(32);
	wMaskBtPanelLeft:WORD;
	wMaskBtPanelRight:WORD;
	wMaskFunctionPanel:WORD;
	wMaskTouchScreenNavPanel:WORD;
	(* process mask *)
	wMaskProcBtPanelLeft:WORD;
	wMaskProcBtPanelRight:WORD;
	wMaskProcFunctionPanel:WORD;
	(* functions *)
	aiRTrigActionPanelLeft:ARRAY[1..5] OF INT:=5(0);
	aiRTrigActionPanelRight:ARRAY[1..5] OF INT:=5(0);
	aiFTrigActionPanelRight:ARRAY[1..5] OF INT:=5(0);
	aiRTrigActionFunctionPanel:ARRAY[1..12] OF INT:=12(0);
	aiRTrigActionTouchScreenNavPanel:ARRAY[1..6,1..9] OF INT;	(* 6 Task und max 9 Seiten pro Task *)
	(* start/stop button *)
	xMaskBtStart:BOOL;
	xMaskBtStop:BOOL;
END_STRUCT
END_TYPE

(* Data type in VISUALISIERUNG *)
TYPE ST_CTRLEACTION :
STRUCT
(* Input *)
	xExecute:BOOL;
	xReset:BOOL;
	iFunction:INT;
	xDeleteVisuFunction:BOOL;		(* Durch setzen dieses Signals wird die aufgerufene Visu Funktion zurückgesetzt *)
	xFunctionActive:BOOL;			(* Visufunktionen, die nicht die Ressource besetzen bestimmen mittels diesem Flag dass die Funktion aktiv ist *)
(* Output *)
	xDone:BOOL;
	xNotReady:BOOL;
	xErr:BOOL;
	udiErrorID:UDINT;
END_STRUCT
END_TYPE

(* Data type in VISUALISIERUNG *)
TYPE ST_CTRLEBUTTON :
STRUCT
	T_Start:ST_BUTTON;
	T_Stop:ST_BUTTON;
	xForceSetStartButton:BOOL;		(* Gilt für Prozess oder Funktionen wo die Starttaste mehrere male gedrückt werden muss *)
	xForceSetStopButton:BOOL;		(* Gilt für Prozess bei Eingabeaufforderung, wo die Schicht 4 noch nicht aktiviert wurde *)
END_STRUCT
END_TYPE

(* Data type in VISUALISIERUNG *)
TYPE ST_CTRLEPROCESS :
STRUCT
(* Input *)
	xExecute:BOOL;
	xReset:BOOL;
	iFunction:INT;
(* Output *)
	xDone:BOOL;
	xErr:BOOL;
	udiErrorID:UDINT;
END_STRUCT
END_TYPE

(* Data type in VISUALISIERUNG *)
TYPE ST_CTRLEVISU :
STRUCT
(* Input *)
	xActive:BOOL;
	xExecute:BOOL;
	xReset:BOOL;
	iFunction:INT;
(* Output *)
	xDone:BOOL;
	xErr:BOOL;
	udiErrorID:UDINT;
	xQvis:BOOL;
END_STRUCT
END_TYPE

(* Data type in VISUALISIERUNG *)
TYPE ST_EXCHG_ANALOGSENSOR :
STRUCT
	rActual_Position:REAL;
	rActual_Offset:REAL;
	rSaved_Position:REAL;
	iSelectHC_Position:INT;
	rMeasureDistance:REAL;
	rScaleFactor:REAL;
END_STRUCT
END_TYPE

(* Data type in VISUALISIERUNG *)
TYPE ST_EXCHG_AXIS :
(*Struct for 'manual' axis-Setup actions from/to HMI *)
STRUCT
	iSetup_AxisSel		:INT:=1;	(*  Achsen; Auswahl 1=Z, 2 & 3=S *)
	arAxis				:ARRAY [1..gcIAxisMax] OF ST_AXIS_LIVESTATE;

	xDisableAxisSelectButton	:BOOL;	(*Betätigung des 'AxisSelect Button' sperren*)
	xJogInc_Common_Setup_Axis		:BOOL;	(*Status zum Umschalten der 'Taskbar right' für Jog oder Ink-->erfolgt über die externe Taste *)
	arTeachSelStep:ARRAY [1..gcIAxisMax] OF REAL;	(*	1=Axis Z Schrittgrösse *)
	arTeachSelVel:ARRAY [1..gcIAxisMax] OF REAL;	(*	1=Axis Z Geschwindigkeit *)
	rTeachSelStep:REAL;	(* Anzeigen der Schrittgrösse der ausgewählten Achse *)
	rTeachSelVel:REAL;	(* Anzeigen der Geschwindigkeit der ausgewählten Achse *)

	arAxisCommon				:ST_AXIS_LIVESTATE;
	rAxisSSpeedCommon:REAL;
	rAxisOSpeedCommon:REAL;
END_STRUCT
END_TYPE

(* Data type in VISUALISIERUNG *)
TYPE ST_EXCHG_BTFUNCTIONPANEL :
STRUCT
	wState:WORD;
	wActivBt:WORD;
	wNotMasktext:WORD;
END_STRUCT
END_TYPE

(* Data type in VISUALISIERUNG *)
TYPE ST_EXCHG_BTPARAMETERLIST :
STRUCT
	wState:WORD;		(* Anzeigen welche Liste ausgewählt ist-->Liste 1-10-->2x1=Liste 1,2x10=Liste 2,2x100=Liste 3 usw. *)
	wActivBt:WORD;		(* Button für Auswahl der Parameterliste-->Liste 1-10-->2x1=Liste 1,2x10=Liste 2,2x100=Liste 3 usw. *)
	wNotMasktext:WORD;	(* Unterdrücken des Textes und disablen des Button der jeweiligen Liste-->Liste 1-10-->2x1=Liste 1,2x10=Liste 2,2x100=Liste 3 usw.-->wenn Bit gesetzt ist, dann wird es unterdrückt *)
	aiSelectText:ARRAY [1..15] OF INT;	(* Für jede Liste kann der entsprechende Text mittels einer definierten Nummer ausgewählt werden*)
	iEditParam:INT;					(* Nummer der anzuzeigenden Parameterliste-->gleiche Nummerierung wie bei aiSelectText *)
	bParameterListEditable:BYTE;		(* 0=unterdrückt die Listen Navigierung für die Auswahl der Parameterliste die Navigierung für die einzelnen Parameter-->Bei Task wo keine Parameterliste besten!
									    1=Parameter Liste ist Editierbar
									    2=Parameter Liste ist nicht Editierbar *)
	bMessageParameter:BYTE;		(* 0=Unterdrücken der Parameter Nachricht, 1=Nur mittels Operator Level, 2=Nur mittels System Level, 3=Keine Parameterliste vorhanden *)
END_STRUCT
END_TYPE

(* Data type in VISUALISIERUNG *)
TYPE ST_EXCHG_CONFIG :
STRUCT
	xNoTouchScreenBtPanel:BOOL;
END_STRUCT
END_TYPE

(* Data type in VISUALISIERUNG *)
TYPE ST_EXCHG_CYLINDER :
STRUCT
	iSelCyl_Setup		:INT;	(*angewählte funktion in Setup Mode , kann als Index verwendet werden für  folgende Statusarray*)
	arStat				:ARRAY [1..7] OF ST_CYLSTAT;
END_STRUCT
END_TYPE

(* Data type in VISUALISIERUNG *)
TYPE ST_EXCHG_FUNCTION_COMMON :
STRUCT
	iFunctionNrMicrohead:INT;	(* 	1=Grundstellungsfahrt BearbStation
									2=S Axis EIN
									3=Wz Einfädeln
									4=Bearbeitungsprozess
									5=S Axis AUS *)
(* Setup Potentiometer *)
	adiPotentiometerValue					:ARRAY [0..11] OF DINT;	(* Wert für Potentiometerstellung *)
END_STRUCT
END_TYPE

(* Data type in VISUALISIERUNG *)
TYPE ST_EXCHG_INFO_PROCESS :
STRUCT
	xOnlineValueModified:BOOL;
	iProfile:INT;
	sProfileName:STRING(30);

	tActualCycleTime:TIME;
	tLastCycleTime:TIME;
	tActualEffProcTime:TIME;
	tLastEffProcTime:TIME;
	rActualFirstContactPosition:REAL;
	rLastFirstContactPosition:REAL;
	rLastOverLimitPosition:REAL;
	rDiffOverLimitPosition:REAL;
	iOverLimitCounter:INT;
	iOverLimitCounterCentering:INT;
	iOverLimitCounterTorque:INT;
	iOverLimitCounterSpeed:INT;							(* IGS *)
	rCuttingSpeed:REAL;
	bLastDetectionSignal:BYTE;	(*	1=< Wz Auslenk. Sensor >
									2=< Wz Drehmom. HC>
									3=< Wz Drehmom. v >
									4=< Wz Auslenk.+Wz Drehm.HC >
									5=< Max. BearbArbeit >	*)
	bPartQuality:BYTE; 	(* 0=Hole not worked, 1=Go HC, 2=Go No HC, 3=NoGo minTime, 4=NoGo maxTime, 5=NoGo insert fail, 6=NoGo NoWP detect, 7=Working, 8=Cycle aborted, 9=No WP, 10=NoGo HC Centr., 11=WP Centered *)

	diWPNumber:DINT;

(* Gilt für die Anzeige der geleisteten Arbeit *)
	rProcessWork:REAL;			(* Bearbeitungsarbeit *)		(* IGS *)
	rActTorque:REAL;										(* IGS *)

	xTorqueLastHC:BOOL;									(* IGS *)
	rTorqueAfterHC_Min:REAL;								(* IGS *)
	rTorqueAfterHC_Max:REAL;								(* IGS *)
	xDeflectionLastHC:BOOL;								(* IGS *)
	rTorqueHC:REAL;										(* IGS *)
	rActualCycleTime:REAL;								(* IGS *)
	rActualEffProcTime:REAL;								(* IGS *)
	iHCTorquePos:INT;									(* IGS *)
	iHCDeflectionPos:INT;									(* IGS *)
	xHCSparkOut:BOOL;									(* IGS *)

	rTorqueMaxAfterWork:REAL;			(* Prozentanzeige des maximalen Drehmoment beim zurückfahren nach der Bearbeitung *)
	rTorqueMaxAfterWorkZPos:REAL;		(* Auf welcher Z Position beim zurückfahren das maximale Drehmoment erreicht wurde *)
END_STRUCT
END_TYPE

(* Data type in VISUALISIERUNG *)
TYPE ST_EXCHG_LAMPTEST :
STRUCT
	xButtonLampIO:BOOL;
	xButtonLampNIO:BOOL;
	xButtonOK:BOOL;
	xShowSelectIONIOButton:BOOL;
	xShowLampTestResult:BOOL;
	sTextLinesEngl:ARRAY [1..18] OF STRING(90);
	sControlMessage1Engl:STRING(90);
	sControlMessage2Engl:STRING(90);
	sTextLines:ARRAY [1..18] OF STRING(90);
	sControlMessage1:STRING(90);
	sControlMessage2:STRING(90);

	abLedControlButton:ARRAY [1..6] OF BYTE;	(*	1=StartButtonLED
													2=StopButtonLED
													3=SetupButtonLED
													4=ReleasButtonLED
													5=SETUPLED
													6=RequestOpenDoorButtonLED
											*)
	abLedStationButton:ARRAY [1..6] OF BYTE;	(*	1=Station1LED
													2=Station2LED
													3=Station3LED
													4=Station4LED
													5=Station5LED
													6=Station6LED
											*)
	abLedControlLamp:ARRAY [1..3] OF BYTE;	(*	1=ControlLampGreen
													2=ControlLampRed
													3=ControlLampYellow
											*)
	abLedSetupLamp:ARRAY [1..2] OF BYTE;	(*	1=SetupLamp1
													2=SetupLamp2
											*)
END_STRUCT
END_TYPE

(* Data type in VISUALISIERUNG *)
TYPE ST_EXCHG_LEVEL :
STRUCT
	iActLevel:INT;
	diPwUser:DINT;
	diPwOperator:DINT:=-1;
	diPwOperatorSaved:DINT;
	diPwSystem:DINT:=-1;
	diRandom:DINT;

	diInputOldPasword:DINT;
	diInputNewPasword:DINT;
	diInputRepeatPasword:DINT;
	xButton_OK:BOOL;
	xButton_Abord:BOOL;
	xShow_Overlay_NewPassword:BOOL;
END_STRUCT
END_TYPE

(* Data type in VISUALISIERUNG *)
TYPE ST_EXCHG_MESSAGE :
STRUCT
	iState:INT;
	iStateBIOS:INT;
	sDynamicTextEnglish:STRING(100);
	sDynamicTextDeutsch:STRING(100);
	sDynamicTextFrancais:STRING(100);
	xShowMessageInfo:BOOL;		(* Zeilenmeldung für Informationen *)
	xShowMessageInput:BOOL;		(* Zeilenmeldung für Eingabeaufforderung *)
	xShowMessageWarning:BOOL;	(* Zeilenmeldung für Warnungen *)
END_STRUCT
END_TYPE

(* Data type in VISUALISIERUNG *)
TYPE ST_EXCHG_MESSAGE_LIST :
STRUCT
	asMsgErrorList:ARRAY [1..20] OF STRING(100);
END_STRUCT
END_TYPE

(* Data type in VISUALISIERUNG *)
TYPE ST_EXCHG_PARAM_AUTOMAT :
STRUCT
(* Gilt für das Aufzeichnen der Zeit des Automatik Prozess *)
	tAutoProcessTime_St1St2:TIME;		(* hh:mm:ss *)
	iAutoProcessDay_St1St2:INT;			(* Anzahl Tage *)
	tActualActiveTime_St1:TIME;	(* hh:mm:ss *)
	iActualActiveTime_St1:INT;		(* Anzahl Tage *)


	diNumberPartWorked_St1St2:DINT;

END_STRUCT
END_TYPE

(* Data type in VISUALISIERUNG *)
TYPE ST_EXCHG_PARAM_AXIS_STATE :
STRUCT
	xReferencedZAxis:BOOL;	(* TRUE= Erstinitialisierung der Z Achse wurde durchgeführt *)

	rPositionReferenceZAxis:REAL;
	rPositionReferenceZAxis_Old:REAL;
	rPositionNegLimitSwitchZAxis:REAL;
	rPositionNegLimitSwitchZAxis_Old:REAL;

	rZDetectEndSwitchSpeed:REAL;
END_STRUCT
END_TYPE

(* Data type in VISUALISIERUNG *)
TYPE ST_EXCHG_PARAM_BIOS :
STRUCT
	xReferencedZAxis_St1:BOOL;	(* TRUE= Erstinitialisierung der Z Achse wurde durchgeführt *)
END_STRUCT
END_TYPE

(* Data type in VISUALISIERUNG *)
TYPE ST_EXCHG_PARAM_CONTRMOT :
STRUCT
	iCurrentReg_PGain:INT;
	iCurrentReg_IGain:INT;
	iSpeedReg_PGain:INT;
	iSpeedReg_IGain:INT;
	iPositionReg_PGain:INT;
	iPositionReg_IGain:INT;
	iPositionReg_DGain:INT;
END_STRUCT
END_TYPE

(* Data type in VISUALISIERUNG *)
TYPE ST_EXCHG_PARAM_CYLINDER :
STRUCT
	rTimeAfterSensorON:REAL;
	rTimeAfterSensorOFF:REAL;
	rTimeOutError:REAL;
	rTimeDelayON:REAL;
	rTimeDelayOFF:REAL;
END_STRUCT
END_TYPE

(* Data type in VISUALISIERUNG *)
TYPE ST_EXCHG_PARAM_ONLINECHANGE :
STRUCT
	T_Data:ST_PROFILEONLINECHANGE_DATA;
	T_DataValPercentAbs:ST_PROFILEONLINECHANGE_DATA;
	T_DataValPercentRel:ST_PROFILEONLINECHANGE_DATA;
	T_Inc:ST_PROFILEONLINECHANGE_DATA;
	T_Max:ST_PROFILEONLINECHANGE_DATA;
	T_Min:ST_PROFILEONLINECHANGE_DATA;
END_STRUCT
END_TYPE

(* Data type in VISUALISIERUNG *)
TYPE ST_EXCHG_PARAM_SPINDLEBURNIN :
STRUCT
	rTimeSpindleActive:REAL;
	rTimeSpindleInactive:REAL;
	rTimeMaxActiveFunction:REAL;
	rSpindleSpeed:REAL;
END_STRUCT
END_TYPE

(* Data type in VISUALISIERUNG *)
TYPE ST_EXCHG_PARAM_SPINDLECALIBRATION :
STRUCT
	arOffsetToolDeflection:ARRAY [1..5] OF REAL;	(* 1=Aktueller Offset, 2=vorgehender Offset usw *)
	arOffsetToolTorque:ARRAY [1..5] OF REAL;	(* 1=Aktueller Offset, 2=vorgehender Offset usw *)
	rEffectiveForceToolDeflection:REAL;
	rNullValueToolDeflection:REAL;
	rEffectiveForceToolTorque:REAL;
	rNullValueToolTorque:REAL;
	iSelectCalibrationCylinder:INT;
END_STRUCT
END_TYPE

(* Data type in VISUALISIERUNG *)
TYPE ST_EXCHG_PARAM_SPINDLESYSTEM :
STRUCT
	rPistonDiameterD1:REAL;		(* the spindle diameter d1 of the ToolDeflection  *)
	rPistonDiameterD2:REAL;		(* the spindle diameter d2 of the Tooldeflection  *)
	rMaxServoAirPressure:REAL;	(* max air pressure of the servo ventil *)
	rMaxDeflectionForce:REAL;		(* calculated max. force of the wire deflection *)
	rMaxServoVoltage:REAL;		(* maximale Ausgangsspannung der Analogen Klemme damit der maximale Druck erreicht wird *)
END_STRUCT
END_TYPE

(* Data type in VISUALISIERUNG *)
TYPE ST_EXCHG_PARAM_SPINDLESYSTEM_L :
STRUCT
	rPistonDiameterD1:REAL;		(* the spindle diameter d1 of the ToolDeflection  *)
	rPistonDiameterD2:REAL;		(* the spindle diameter d2 of the Tooldeflection  *)
	rMaxServoAirPressure:REAL;	(* max air pressure of the servo ventil *)
	rMaxDeflectionForce:REAL;		(* calculated max. force of the wire deflection *)
	rMaxServoVoltage:REAL;		(* maximale Ausgangsspannung der Analogen Klemme damit der maximale Druck erreicht wird *)
END_STRUCT
END_TYPE

(* Data type in VISUALISIERUNG *)
TYPE ST_EXCHG_PARAM_STANDARDPROCESS :
STRUCT
(* Position *)
	rPositionLoad:REAL;
	rPositionStartProc:REAL;
	rPositionEndProc:REAL;
	rPositionEndMech:REAL;
	rPositionToolChange:REAL;
	iHCStartProcPosCounter:INT;
(* Infeed Tool *)
	rInfeedZAxisSpeed:REAL;
	rInfeedSpindleSpeed:REAL;
	iNumberTryInfeed:INT;
	rInfeedOffsetBackward:REAL;
	rInfeedForceDeflection:REAL;
(* Spark out *)
	rSparkOutStrokeLength:REAL;
	iSparkOutStrokeCount:INT;
	rSparkOutStrokeSpeed:REAL;
	rSparkOutForceDeflection:REAL;
	rSparkOutTorqueLevel:REAL;		(* Schwellwert für Drehmoment beim Ausfunken-->für HC *)
(* Process time *)
	rProcessMinTime:REAL;
	rProcessMaxTime:REAL;
(* Outfeed *)
	rOutfeedStrokeAxisSpeed:REAL;
	rOutfeedSpindleSpeed:REAL;
(* Neu nicht mehr als OnlineChange Parameter definiert *)
	rDeflectionSensorOffset:REAL;
(* Drehmomentüberlast *)
	rTorqueLevel_Overload:REAL;
(* Progressiv Stroke *)
	rDistProgressStroke:REAL; 			(* [mm] Vertikale Distanz, welche das Intervall zwischen den Rückzieher definiert *) (* BEF *)
	iProgressStrokeStartTorque:INT; 	(* [%] Notwendiges Drehmoment um den ersten Rückhub zu erzwingen und somit die progressive Hubfunktion zu starten. In Prozent bezogen auf das Hard Contact Drehmoment («WzDrehm. HC») *) (* BEF *)
(* Abblasdüse *)
	iCleanNozzleMode:INT; 			(*0=Duese nicht eingeschaltet,1= für positive Z1 Geschwindigkeiten eingeschaltet, 2=für negative Z1 Geschwindigkeiten eingeschaltet, 3=für jegliche Geschwindigkeiten eingeschaltet *) (* BEF *)
(* Positionen *)
	rPosToolGuid_Up:REAL;			(* Position des Schlitten des oberen Führungsrohr auf der oberen Position *)
	rPosToolGuid_Down:REAL;			(* Position des Schlitten des oberen Führungsrohr auf der untere Position *)
	rDistanceToolGuide:REAL;			(* Abstand zwischen dem unteren Führungsrohr und der Lufttischplatte *)
	rDistanceToolEndPos:REAL;		(* Abstand zwischen der Luft Tischplatte und der Werkzeug End Position *)
	rLengthTool_Fixed:REAL;			(* Einspannlänge *)
	rLengthTool_Work:REAL;			(* Bearbeitungslänge *)
	rLengthToolGuide:REAL;			(* Länge des oberen Führungsrohreinsatz *)
	rLengthAirTableBoard:REAL;		(* Höhe der Lufttischplatte gemessen von der Tischplatte aus *)
	xConfigActive:BOOL;				(* TRUE=Positionen der Z Achse mittel der Konfigurationswerte, FALSE=Positionen der Z Achse mittels getachte Werte *)

	iMaxTorque:INT;																									(* IGS *)
	rSpeedZAxisForBackward:REAL;	(* Z1 Geschwindigkeit, falls diese erreicht wird das künstlich ein Rückhub erzwingt wird *)		(* IGS *)
	rWorkingSpeedOscillation:REAL;																					(* IGS2 *)
	rZ1AxisPosSwitchOAxisOff:REAL;	(* Ausschaltpunkt für die O-Achse (Schnellhub) *)										(* IGS2 *)
	xActivateCoolantProcess:BOOL;																						(* IGS2 *)
	rStrokeAxisPosSwitchCoolantOff:REAL;																				(* IGS2 *)
(* Zentrieren *)
	rCentringPosZ1Axis:REAL;					(* Z1 Achse ZentrierPosition *)																(* IGS3 *)
	rCentringPosSpeedSlowZ1Axis:REAL;		(* Z1 Achse langsame Geschwindigkeit während dem Zentrieren *)								(* IGS3-->PUM: Name geändert *)
	rCentringPosSpeedFastZ1Axis:REAL;			(* Z1 Achse schnelle Geschwindigkeit während dem Zentrieren *)								(* PUM: Neu für Zentrierprozess *)
	rCentringSpeedSAxis:REAL;					(* S Achse Drehzahl während dem Zentrieren *)												(* IGS3 *)
	rCentringSpeedOAxis:REAL;					(* O Achse Geschwindigkeit während dem Zentrieren *)										(* IGS3 *)
	rCentringBackStrokeOffsetFirstHC:REAL;		(* Z1 Achse Rückhub Offset beim ersten HC während dem Zentrieren *)							(* IGS3-->PUM: Name geändert *)
	rCentringBackStrokeOffsetAfterFirstHC:REAL;	(* Z1 Achse Rückhub Offset nach dem ersten HC während dem Zentrieren *)					(* PUM: Neu für Zentrierprozess *)
	rCentringOffsetBeforeLastHC:REAL;			(* Z1 Achse zum letzten HC minus diesen Offset schnell anfahren während dem Zentrieren *)		(* PUM: Neu für Zentrierprozess *)
	rCentringBackStrokeSpeed:REAL;			(* Z1 Achse Rückhub Geschwindigkeit während dem Zentrieren *)								(* IGS3 *)
	rCentringTimeHCActive:REAL;				(* Ab dem ersten HC bei den nächsten HC wie lange maximal gewartet werden soll wenn der neue Auslenksensor angibt bis ein Rückhub erfolgen soll *)	(* PUM: Neu für Zentrierprozess *)
	rCentringTimeHCInactive:REAL;				(* Ab dem ersten HC bei den nächsten HC wie lange der neue Auslenksensor nicht mehr angeben soll bis es wieder langsam nach vorne fährt *)			(* PUM: Neu für Zentrierprozess *)
	iCentringNumberMaxHCinWindow:INT;		(* Anzahl HC im definierten Fenster die auftreten können bis nIO während dem Zentrieren *)		(* IGS3-->PUM: Neue definition *)
	rCentringHCWindow:REAL;					(* Fenster als Überwachung beim eintreffen der HC wie oft maximal in diesem Fenster eintreffen darf bis nIO während dem Zentrieren *)					(* PUM: Neu für Zentrierprozess *)
	rCentringForceDeflection:REAL;				(* Auslenk Kraft während dem Zentrieren *)													(* IGS3 *)
	rCentringOffsetBackward:REAL;				(* bei erreichen von ZentrierPos einen Offset zurück fahren *)									(* IGS3 *)
	rCenteringDeflectionSensorOffset:REAL;		(* Offset nach welchen Z Fahrweg der HC erst angeben darf *)									(* PUM: Neu für Zentrierprozess *)
	rCentringOffsetSlowToFastZSpeed:REAL;		(* Wie lange maximal die Z Achse beim zentrieren langsam fahren soll bis es auf die schnelle Geschwindigkeit schaltet *)	(* PUM: Neu für Zentrierprozess *)
	iCentringSelectProcess:INT;					(* 1=Konventioneller Zentrier Ablauf, 2=Ablauf mit Grauzone finden *)
(* Suspenstion *)
	rSuspensionBubblerSpeed:REAL;	(* Suspension DC Motor Rührer Geschwindigkeit *)										(* IGS3 *)
	rSuspensionFeederSpeed:REAL;	(* Suspension DC Motor Pumpe Geschwindigkeit *)										(* IGS3 *)
(* Neue Parameter für das Inkrementieren der Z1 EndPosition *)
	xPositionEndProcIncOnOff:BOOL;		(* Hier kann definiert werden ob die Inkrementierung Aktiv sein soll oder nicht. Wenn Wert 0 eingestellt ist, dann ist es wie gehabt *)
	rPositionEndProcMaxInc:REAL;	(* Die Maximale EndPosition die nicht überschritten werden darf beim Inkrementieren der Z1 Position nach jeder Bearbeitung *)
	rPositionEndProInc:REAL;			(* Um wie viel nach jeder Bearbeitung die Z1 EndPosition inkrementiert werden muss *)

(* Neue Reglertype für den Bearbeitungsprozess *)
	iWorkControlType:INT;	(* 0,1=konventionell, 2=Adaptive Vorschubsteuerung mit PID, 3=konevntionell mit PD Regler *)
	(* PID Regler für adaptive Vorschubsteuerung *)
	rZ_PID_Torque:REAL;
	rZ_PID_MinSpeed:REAL;
	rZ_PID_MaxSpeed:REAL;
	rZ_PID_Kp:REAL;
	rZ_PID_Ki:REAL;
	rZ_PID_Kd:REAL;
	iZ_PID_FilterM:INT;
	(* D Regler für konventioneller Regler *)
	rZ_D_Kd:REAL;
	iZ_D_FilterM:INT;

	rOutfeedStrokeAxisSpeedSlow:REAL;		(* Neuer Parameter für das zurückfahren am Prozessende wo man eine langsame Geschwindigkeit definieren kann und nach dem abfahren des Offset mit der normalen Geschwindigkeit zurückfährt *)
	rZ1AxisPosSwitchFastVel:REAL;			(* Neuer Parameter für das zurückfahren am Prozessende nach welcher Z1 Position dann mit der schnellen Geschwindigkeit umstellen soll *)
	rZ1AxisOffsetStartRecordTorque:REAL;		(* Neuer Parameter für das zurückfahren am Prozessende nach welcher Z1 Position die Aufzeichnung für das maximale Drehmoment gestartet werden soll *)

(* Neue Parameter für das Inkrementieren der Z1 Zentrier Position *)
	xCentringEndProcIncOnOff:BOOL;		(* Hier kann definiert werden ob die Inkrementierung in der Zentrierung Aktiv sein soll oder nicht. Wenn Wert 0 eingestellt ist, dann ist es wie gehabt *)
	rCentringEndProInc:REAL;				(* Um wie viel nach jeder Zentrierung die Z1 EndPosition inkrementiert werden muss *)

(* Neue Parameter für den Regler für die Spindel S Achse und der O Achse *)
	rWorkingSpindleSpeedMinMax:REAL;	(* Spindel Regler ist Aktiv wenn dieser Wert nicht gleich Null ist *)
	rO_Ctrl_TorquePercent_OFF:REAL;	(* Schnellhub Regler --> Wenn dieser Schwellwert des Drehmomentes erreicht wird, dann wird der Schnellhub ausgeschaltet und mittels der Hilfe der Hysterese Offset wieder eingeschaltet wird *)
	rO_Ctrl_HystereseOffset:REAL;		(* Schnellhub Regler Aktiv wenn dieser Parameter nicht den Wert Null ist. Ist der Wert Positiv, dann muss das Drehmoment ansteigen damit es den Schnellhub wieder einschaltet. Wert Negativ dann muss es abklingen damit es wieder einschaltet *)

(* Neue Parameter für Abbruchkriterium für den Zylindrischen Bereich *)
	rZPositionCylindricalArea:REAL;			(* Hier bestimmt man für die Z Achse wo der Zylindrische Bereich des Werkzeuges anfängt. Wenn der Wert Null beträgt dann gilt der konventionelle Ablauf *)
	rZMinThresholdTroqueEndProcess:REAL;	(* Hier gibt man den Schwellwert an wo unterschritten werden muss wenn die Z Achse im zylindrischen Bereich ist wo dann als Prozessende gilt *)
	rZPositionCylindricalAreaStop:REAL;		(* Auf welcher Z Position im zylindrischen Bereich der Schwellwert unterschritten wurde *)
END_STRUCT
END_TYPE

(* Data type in VISUALISIERUNG *)
TYPE ST_EXCHG_PARAM_SYSTEM :
STRUCT
	xActive_ProfilLoadNormalMode:BOOL;
	xDataFileActive:BOOL;
	iMachineNumber:INT;
END_STRUCT
END_TYPE

(* Data type in VISUALISIERUNG *)
TYPE ST_EXCHG_PARAM_TEACHIN :
STRUCT
	rIncSlow:REAL;
	rIncFast:REAL;
	rVelSlow:REAL;
	rVelFast:REAL;
	rRefPosition:REAL;
	rRefSpeed:REAL;
	rPositionSpeed:REAL;
	rAcceleration:REAL;
	rDeceleration:REAL;
	rJerk:REAL;
	rDecelerationEmergency:REAL;
	rJerkEmergency:REAL;
	xResetActiveTime: BOOL;
END_STRUCT
END_TYPE

(* Data type in VISUALISIERUNG *)
TYPE ST_EXCHG_PARAM_TOOLCOUNTER :
STRUCT
	diMaxNumberToolCycle:DINT;			(* Max Anz. WzZyklen *)
	diToolCycleCounter:DINT;				(* WzZyklen Zählerstand *)
	diWarningAtToolCycleCounter:DINT;		(* Warnung bei Zählerstand *)
END_STRUCT
END_TYPE

(* Data type in VISUALISIERUNG *)
TYPE ST_EXCHG_PARAM_TORQUESYSTEM :
STRUCT
	rGearRatioGearBox:REAL;					(* Übersetzungsverhältnis des Differentialgetriebe *)
	rPlanetCarrier_Radius:REAL;				(* Radius des Planetenträger *)
	rGearRatioRocker:REAL;					(* Übersetzungsverhältnis der Wippe *)
	rGearRatioSpindleMotor:REAL;				(* Übersetzungsverhältnis des Motorgetriebe *)

	rPistonTorqueHC:REAL;					(* Kolbendurchmesser für HC Drehmoment *)
	rMaxServoAirPressure_HC:REAL;			(* max air pressure of the servo ventil *)
	rMaxServoVoltage_HC:REAL;				(* maximale Ausgangsspannung der Analogen Klemme damit der maximale Druck erreicht wird *)
	rMaxTorque_HC:REAL;					(* calculated max. force of the tool torque *)

	rPistonTorqueHCOverload:REAL;			(* Kolbendurchmesser für HC Überlast Drehmoment *)
	rMaxServoAirPressure_HCOver:REAL;		(* max air pressure of the servo ventil *)
	rMaxServoVoltage_HCOver:REAL;			(* maximale Ausgangsspannung der Analogen Klemme damit der maximale Druck erreicht wird *)
	rMaxTorque_HCOver:REAL;				(* calculated max. force of the tool torque *)

(* Parameter für analoger Drehmomentsensor *)
	rTorquePosition_HC:REAL;
	rTorquePosition_HCOverload:REAL;
	rTorqueScaleFactor:REAL;
	rMeasureDistance:REAL;

	rActual_Torque:REAL;						(* Aktuelles Drehmoment der Drehmomentfeder in mNm *)			(* IGS *)
	rMaxTorque:REAL;						(* Berechnete maximales Drehmoment in mNm *)					(* IGS *)
END_STRUCT
END_TYPE

(* Data type in VISUALISIERUNG *)
TYPE ST_EXCHG_PARAM_TORQUESYSTEM_L :
STRUCT
	rActual_Torque:REAL;						(* Aktuelles Drehmoment der Drehmomentfeder in mNm *)			(* IGS *)
	rMaxTorque:REAL;						(* Berechnete maximales Drehmoment in mNm *)					(* IGS *)

	rMinTorqueLevel:REAL;					(* Drehmoment dass gemessen werden muss, welches den Nullpunkt oder resp. den minimale Drehmoment ergibt *)
END_STRUCT
END_TYPE

(* Data type in VISUALISIERUNG *)
TYPE ST_EXCHG_PARAM_WPCOUNTER :
STRUCT
	diWPCounter_IO_NIO:DINT;		(* WstkZähler tagesaktuell (iO+niO) *)
	diWPCounter_IO_Actual:DINT;	(* WstkZähler tagesaktuell (iO) *)
	diWPCounter_IO_Reset:DINT;	(* WstkZähler rücksetzbar (iO) *)
	diWPCounter_NIO_Actual:DINT;	(* WstkZähler tagesaktuell (niO) *)
	diWPCounter_NIO_Reset:DINT;	(* WstkZähler rücksetzbar (niO) *)
END_STRUCT
END_TYPE

(* Data type in VISUALISIERUNG *)
TYPE ST_EXCHG_PARAM_Z_TGUIDE :
STRUCT
	rOffset_Z_ToolGuide:REAL;				(* Offset für die Abhängigkeit zwischen der Z Achse und dem Massstab des oberen Führungsrohr zu bestimmen *)
	rOffset_Z_ToolGuide_Old:REAL;			(* Offset für die Abhängigkeit zwischen der Z Achse und dem Massstab des oberen Führungsrohr zu bestimmen-->vorheriger Wert *)
	rDistanceTGuideToTableBoard:REAL;	(* Distanz zwischen der Platte des oberen Führungsrohr und der Tischplatte *)
	rScaleDefinedPos:REAL;					(* Definierte Position des Massstabes *)
	rToolLengthSetup:REAL;					(* Werkzeuglänge für die Einrichtung um den Offset zu bestimmen *)
	rDistanceTGuideToTableBoardLess:REAL;	(* Distanz zwischen oberen Führungsrohr und der Tischplatte *)
END_STRUCT
END_TYPE

(* Data type in VISUALISIERUNG *)
TYPE ST_EXCHG_PARTQUALITY :
STRUCT
	bPartQualityStation: BYTE;				(* 0=Hole not worked, 1=Go HC, 2=Go No HC, 3=NoGo minTime, 4=NoGo maxTime, 5=NoGo insert fail, 6=NoGo NoWP detect, 7=Working, 8=Cycle aborted, 9=No WP, 10=NoGo HC Centr., 11=WP Centered *)
	rActualFirstHCPositionStation:REAL;
	iHCCounterStation: INT;
	iHCCounterCenteringStation: INT;
	iHCCounterTorqueStation: INT;
	iHCCounterSpeedStation: INT;			(* IGS *)
	tCycleTimeStation: TIME;
	tWorkTimeStation: TIME;
	bInfeedCounterZ:BYTE;				(* Anzahl Einfädelversuche mit der Z Achse. Wenn erste mal durchgeht dann steht eine 1, wenn erst beim zweiten Versuch dann eine 2 usw. *)

	diActual_NumberHoleToWork:DINT;		(* Aktuell zu bearbeitende Bohrungsnummer *)
	sFileName:STRING(28);				(* Aktuelle Dateiname *)
END_STRUCT
END_TYPE

(* Data type in VISUALISIERUNG *)
TYPE ST_EXCHG_PROFILE_COMMON :
STRUCT
(* State *)
	xImportProzessData:BOOL:=FALSE;
(* Array *)
	T_Id:ST_PROFILE_ID;
	T_ProfileManage:ST_PROFILE_LIST_MANAGE;
	T_ProfileList:ARRAY[1..5] OF ST_PROFILE_LIST;
	T_OnlineChange:ST_EXCHG_PARAM_ONLINECHANGE;
END_STRUCT
END_TYPE

(* Data type in VISUALISIERUNG *)
TYPE ST_EXCHG_SAFETY_CTRL :
STRUCT
	bStateMessageError:BYTE;
	bStateMessageInfo:BYTE;
	bStateMessageWarning:BYTE;
	bStateMessagePreWarning:BYTE;
	bStateMessageRequest:BYTE;
	xMessageActive:BOOL;		(* IGS sobald eine Overlay MessageBox aktiv ist, wird diese Variable TRUE *)
	xConfirmMsgError:BOOL;
	xConfirmMsgInfo:BOOL;
	xConfirmMsgWarning:BOOL;
	xConfirmMsgPreWarning:BOOL;
	xConfirmMsgRequest:BOOL;
	xConfirmMsgPartNumber:BOOL;
	xResetMsgPreWarning:BOOL;
	iMsgErrorLine1:INT;
	iMsgErrorLine2:INT;
	iMsgErrorLine3:INT;
	iMsgErrorLine4:INT;
	iMsgWarningLine1:INT;
	iMsgWarningLine2:INT;
	iMsgWarningLine3:INT;
	iMsgWarningLine4:INT;
	iMsgInfoLine1:INT;
	iMsgInfoLine2:INT;
	iMsgInfoLine3:INT;
	iMsgInfoLine4:INT;
	sDynMsgPreWarningLine1Engl:STRING(55);
	sDynMsgPreWarningLine2Engl:STRING(55);
	sDynMsgPreWarningLine3Engl:STRING(55);
	sDynMsgPreWarningLine4Engl:STRING(55);
	sDynMsgPreWarningLine5Engl:STRING(55);
	sDynMsgPreWarningLine1Ger:STRING(55);
	sDynMsgPreWarningLine2Ger:STRING(55);
	sDynMsgPreWarningLine3Ger:STRING(55);
	sDynMsgPreWarningLine4Ger:STRING(55);
	sDynMsgPreWarningLine5Ger:STRING(55);
	xReadNextPreWarningMessage:BOOL;
	xReadPreviousPreWarningMessage:BOOL;
	xSelect_ToolChange_St1:BOOL;
	bState_Select_St1:BYTE;	(* 1= Station 1 für Wz Wechsel Zähler zurücksetzen ausgewählt *)

